# B&R Automation Studio project TD52 (part 75)

```c
  /* End of Switch: '<S7>/Switch3' */

  /* S-Function (bur_bus_in): '<Root>/Bus Input1' */
  LX2_B.BusInput1 = inst->PERM;

  /* BusSelector: '<S5>/Bus Selector7' */
  rtb_rLX2_inLimitSetup_Time = LX2_B.BusInput1.rLX2_inLimitSetup_Time;

  /* Gain: '<S7>/Gain3' incorporates:
   *  BusSelector: '<S5>/Bus Selector7'
   *  DataTypeConversion: '<S7>/Data Type Conversion2'
   *  Product: '<S7>/RateLimit_multiplier'
   */
  rtb_Gain3 = rtb_Switch7 * (real32_T)LX2_B.BusInput1.iCtrl_RateLimit_TraceBack *
    0.001F;

  /* Product: '<S41>/delta rise limit' incorporates:
   *  SampleTimeMath: '<S41>/sample time'
   *
   * About '<S41>/sample time':
   *  y = K where K = ( w * Ts )
   */
  rtb_Switch2_kt = rtb_Gain3 * 0.1F;

  /* UnitDelay: '<S7>/Unit Delay3' */
  rtb_UnitDelay3 = LX2_DWork.UnitDelay3_DSTATE;

  /* S-Function (bur_bus_in): '<Root>/Bus Input2' */
  LX2_B.BusInput2 = inst->PARA;

  /* BusSelector: '<S51>/Bus Selector4' */
  rtb_rPr_Leanox_Dev = LX2_B.BusInput.rPr_Leanox_Dev;
  rtb_rP_Set_Norm = LX2_B.BusInput.rP_Set_Norm;

  /* BusSelector: '<S51>/Bus Selector5' */
  rtb_iFiltConst_LeanoxDev_Steady =
    LX2_B.BusInput1.iFiltConst_LeanoxDev_SteadyState;
  rtb_iFiltConst_P_set_SteadyStat = LX2_B.BusInput1.iFiltConst_P_set_SteadyState;

  /* Logic: '<S51>/Logical Operator1' */
  rtb_LogicalOperator1 = !LX2_B.BusInput.bLX2_active;

  /* Outputs for Atomic SubSystem: '<S51>/Filter' */
  LX2_Filter1(rtb_iFiltConst_LeanoxDev_Steady, rtb_LogicalOperator1,
              rtb_rPr_Leanox_Dev, &LX2_B.Filter, &LX2_DWork.Filter, inst);

  /* End of Outputs for SubSystem: '<S51>/Filter' */

  /* RelationalOperator: '<S51>/ ' incorporates:
   *  Abs: '<S51>/Abs'
   *  Product: '<S51>/Thres'
   */
  rtb_u = ((real32_T)fabs(LX2_B.Filter.Switch) <=
           LX2_B.BusInput1.rThreshold_LeanoxDev_SteadyState *
           LX2_B.BusInput2.rLX2_SteadyStateFactor);

  /* Logic: '<S51>/Logical Operator3' */
  rtb_LogicalOperator3 = !LX2_B.BusInput.bLX2_active;

  /* Outputs for Atomic SubSystem: '<S51>/Filter1' */
  LX2_Filter1(rtb_iFiltConst_P_set_SteadyStat, rtb_LogicalOperator3,
              rtb_rP_Set_Norm, &LX2_B.Filter1, &LX2_DWork.Filter1, inst);

  /* End of Outputs for SubSystem: '<S51>/Filter1' */

  /* Sum: '<S51>/Sum2' */
  rtb_Switch7 = LX2_B.Filter1.Switch - rtb_rP_Set_Norm;

  /* Abs: '<S51>/Abs1' */
  rtb_Switch7 = (real32_T)fabs(rtb_Switch7);

  /* RelationalOperator: '<S51>/   ' incorporates:
   *  Product: '<S51>/Thres1'
   */
  rtb_u_b = (rtb_Switch7 <= LX2_B.BusInput1.rThreshold_P_set_SteadyState *
             LX2_B.BusInput2.rLX2_SteadyStateFactor);

  /* Logic: '<S51>/Logical Operator2' incorporates:
   *  Logic: '<S51>/Logical Operator4'
   */
  rtb_LogicalOperator2 = (LX2_B.BusInput.bLX2_active && rtb_u && rtb_u_b &&
    (!LX2_B.BusInput.bExt_SteadyState_Loss));

  /* Outputs for Atomic SubSystem: '<S51>/TON' */
  /* Logic: '<S59>/Logical Operator2' */
  rtb_LogicalOperator2_de = !rtb_LogicalOperator2;

  /* DiscreteIntegrator: '<S59>/Discrete-Time Integrator' */
  if (rtb_LogicalOperator2_de || (LX2_DWork.DiscreteTimeIntegrator_PrevRe_m != 0))
  {
    LX2_DWork.DiscreteTimeIntegrator_DSTATE_l = 0U;
  }

  /* RelationalOperator: '<S59>/Relational Operator' incorporates:
   *  DiscreteIntegrator: '<S59>/Discrete-Time Integrator'
   */
  tmp_0 = (uint32_T)LX2_DWork.DiscreteTimeIntegrator_DSTATE_l * 52429U;
  rtb_RelationalOperator_b = (((tmp_0 & 4U) != 0U) + (tmp_0 >> 3) >= ((uint32_T)
    LX2_B.BusInput1.iTiDelay_SteadyState << 16));

  /* Logic: '<S59>/Logical Operator3' */
  rtb_LogicalOperator3_e = (rtb_RelationalOperator_b && rtb_LogicalOperator2);

  /* Update for DiscreteIntegrator: '<S59>/Discrete-Time Integrator' incorporates:
   *  Logic: '<S59>/Logical Operator'
   *  Logic: '<S59>/Logical Operator1'
   */
  LX2_DWork.DiscreteTimeIntegrator_DSTATE_l = (uint16_T)((uint32_T)
    ((!rtb_RelationalOperator_b) && rtb_LogicalOperator2) + (uint32_T)
    LX2_DWork.DiscreteTimeIntegrator_DSTATE_l);
  if (rtb_LogicalOperator2_de) {
    LX2_DWork.DiscreteTimeIntegrator_PrevRe_m = 1;
  } else {
    LX2_DWork.DiscreteTimeIntegrator_PrevRe_m = 0;
  }

  /* End of Update for DiscreteIntegrator: '<S59>/Discrete-Time Integrator' */
  /* End of Outputs for SubSystem: '<S51>/TON' */

  /* MATLAB Function: '<S8>/MATLAB Function' incorporates:
   *  Constant: '<S65>/Constant'
   *  Logic: '<S52>/Logical Operator'
   *  Logic: '<S52>/Logical Operator10'
   *  RelationalOperator: '<S65>/Compare'
   */
  /* MATLAB Function 'Leanox 2.0/STM/MATLAB Function': '<S53>:1' */
  /* % Header */
  /*  This Function controls the features of LX2, like saving the map, gasmixing, enabling/disabling, timer, etc., */
  /*  depending on various inputs. */
  /*  Rev 1 : Christian Schneider, 24.08.2018 */
  /*  Rev 1.1 : Enrico Maran, 17.10.2019, Removed bLeanox_Adjust input/use */
  /*  Rev 1.2 : Enrico Maran, 17.02.2021, Removed closed loop freezing if bEng_misfire; added external interface for BPOC learning stop */
  /*  */
  /* % LX2 State Machine */
  /*  -> LEANOX 2.0 is OFF */
  if ((!LX2_B.BusInput2.bLX2_enable) || (!LX2_B.BusInput.bLX2_active)) {
    /*  LX2 off */
    /*  function undesired_operating */
    /* % function my_gasmixing <<LX2_FunReq-26>> */
    /*  define output vectors */
    /*  undefined Gastype */
    rtb_splitfactor_Gas[0] = 0.0F;
    rtb_splitfactor_Gas[1] = 0.0F;
    rtb_splitfactor_Gas[2] = 0.0F;
    rtb_splitfactor_Gas[3] = 0.0F;
    tmp[0] = 1.0F;
    tmp[1] = 1.0F;
    LX2_my_BPOC_enable_h(rtb_splitfactor_Gas, FALSE, tmp,
                         LX2_B.BusInput.bExt_BPOC_learning_Stop,
                         rtb_bBPOC_enable_a, rtb_bSave_BPOC_enable, inst);
    bCtrl_enable = FALSE;

    /*  NOx controler enable */
    bCtrl_freeze = TRUE;

    /*  freeze NOx controler output */
    b_bEng_knock = FALSE;
    bEng_misfire = FALSE;

    /*  -> LEANOX 2.0 is ON */
  } else if ((!LX2_B.BusInput.bLeanox_Engine_Man) && (rtb_LogicalOperator3_e &&
              LX2_B.BusInput.bNOx_valid && (!LX2_B.BusInput.bESC_active) &&
              (LX2_B.BusInput.rNOx_act >= 10.0F))) {
    /*  Engine in Leanox Auto Mode */
    /*              bBPOC_enable_Gas1=true;  */
    /*              bSave_BPOC_enable_Gas1=true; */
    LX2_my_gasmixing(LX2_B.BusInput.iIdx_Gtyp_Dem,
                     LX2_B.BusInput.rGT_QualMix_1_2, LX2_B.BusInput.rGT_RatioMix,
                     TRUE, LX2_B.BusInput1.rThreshold_save2map,
                     LX2_B.BusInput.bExt_BPOC_learning_Stop, rtb_splitfactor_Gas,
                     rtb_bBPOC_enable_a, rtb_bSave_BPOC_enable, inst);
    bCtrl_enable = TRUE;

    /* % function Misfire and Knocking handlig at LX2 */
    if (LX2_B.BusInput.rKnock_level <= LX2_B.BusInput1.rThreshold_knock) {
      b_bEng_knock = FALSE;
    } else {
      b_bEng_knock = TRUE;
    }

    if (LX2_B.BusInput.rMisfire_level <= LX2_B.BusInput1.rThreshold_misfire) {
      bEng_misfire = FALSE;
    } else {
      bEng_misfire = TRUE;
    }

    bCtrl_freeze = b_bEng_knock;
  } else {
    /*  Engine in Leanox Manuel Mode >or< not allowed to act -> freeze output of LX2 and do not update BPOC */
    LX2_my_gasmixing(LX2_B.BusInput.iIdx_Gtyp_Dem,
                     LX2_B.BusInput.rGT_QualMix_1_2, LX2_B.BusInput.rGT_RatioMix,
                     FALSE, LX2_B.BusInput1.rThreshold_save2map,
                     LX2_B.BusInput.bExt_BPOC_learning_Stop, rtb_splitfactor_Gas,
                     rtb_bBPOC_enable_a, rtb_bSave_BPOC_enable, inst);
    bCtrl_enable = FALSE;
    bCtrl_freeze = TRUE;
    b_bEng_knock = FALSE;
    bEng_misfire = FALSE;
  }

  /* Switch: '<S7>/Switch7' incorporates:
   *  Gain: '<S7>/mbar2bar1'
   *  MATLAB Function: '<S8>/MATLAB Function'
   */
  /* '<S53>:1:4' */
  if (bEng_misfire) {
    rtb_Switch7 = rtb_UnitDelay3;
  } else {
    rtb_Switch7 = 0.001F * LX2_B.BusInput2.rPr_LX2_OffsetLimit;
  }

  /* End of Switch: '<S7>/Switch7' */

  /* BusSelector: '<S5>/Bus Selector2' */
  rtb_Switch_nq = LX2_B.BusInput2.rLX2_Ctrl_Tn;

  /* RelationalOperator: '<S32>/Compare' incorporates:
   *  BusSelector: '<S5>/Bus Selector2'
   *  Constant: '<S32>/Constant'
   */
  rtb_Compare_n = (LX2_B.BusInput2.rLX2_Ctrl_Tn <= 0.0F);

  /* BusSelector: '<S5>/Bus Selector4' */
  rtb_rNOx_act_g = LX2_B.BusInput.rNOx_act;

  /* Logic: '<S5>/Logical Operator6' */
  rtb_LogicalOperator6_a = !LX2_B.BusInput.bLX2_active;

  /* UnitDelay: '<S7>/Unit Delay1' */
  rtb_UnitDelay1 = LX2_DWork.UnitDelay1_DSTATE;

  /* Logic: '<S52>/Logical Operator11' incorporates:
   *  Logic: '<S52>/Logical Operator5'
   *  Logic: '<S52>/Logical Operator6'
   *  Logic: '<S52>/Logical Operator7'
   *  Logic: '<S52>/Logical Operator8'
   *  UnitDelay: '<S52>/Unit Delay1'
   */
  rtb_LogicalOperator_f = (LX2_DWork.UnitDelay1_DSTATE_l ||
    (((!LX2_B.BusInput2.bLX2_enable) || (!LX2_B.BusInput.bLX2_active)) &&
     LX2_B.BusInput.bBPOC_reset));

  /* Logic: '<S54>/Logical Operator4' incorporates:
   *  Logic: '<S54>/Logical Operator1'
   *  Logic: '<S54>/Logical Operator27'
   *  Logic: '<S54>/Logical Operator3'
   *  UnitDelay: '<S54>/Unit Delay'
   */
  rtb_LogicalOperator4_n = ((!LX2_DWork.UnitDelay_DSTATE_l) &&
    (!rtb_LogicalOperator_f) && (rtb_bSave_BPOC_enable[0] ||
    rtb_bSave_BPOC_enable[1] || rtb_bSave_BPOC_enable[2] ||
    rtb_bSave_BPOC_enable[3]));

  /* DataTypeConversion: '<S54>/Data Type Conversion' incorporates:
   *  BusSelector: '<S54>/Bus Selector5'
   */
  rtb_DataTypeConversion = (real32_T)LX2_B.BusInput1.iTiUpdate_BPOC;

  /* Outputs for Atomic SubSystem: '<S54>/TON' */
  LX2_TON(rtb_LogicalOperator4_n, rtb_DataTypeConversion, &LX2_B.TON_p,
          &LX2_DWork.TON_p, inst);

  /* End of Outputs for SubSystem: '<S54>/TON' */

  /* Switch: '<S54>/Switch2' incorporates:
   *  Switch: '<S54>/Switch1'
   */
  if (rtb_LogicalOperator_f) {
    rtb_Switch2_a_idx = TRUE;
    rtb_Switch2_a_idx_0 = TRUE;
    rtb_Switch2_a_idx_1 = TRUE;
    rtb_Switch2_a_idx_2 = TRUE;
  } else if (LX2_B.TON_p.LogicalOperator3) {
    /* Switch: '<S54>/Switch1' */
    rtb_Switch2_a_idx = rtb_bSave_BPOC_enable[0];
    rtb_Switch2_a_idx_0 = rtb_bSave_BPOC_enable[1];
    rtb_Switch2_a_idx_1 = rtb_bSave_BPOC_enable[2];
    rtb_Switch2_a_idx_2 = rtb_bSave_BPOC_enable[3];
  } else {
    rtb_Switch2_a_idx = FALSE;
    rtb_Switch2_a_idx_0 = FALSE;
    rtb_Switch2_a_idx_1 = FALSE;
    rtb_Switch2_a_idx_2 = FALSE;
  }

  /* End of Switch: '<S54>/Switch2' */

  /* Gain: '<S8>/Gain7' */
  rtb_Gain7 = 100.0F * LX2_B.BusInput.rP_Set_Norm;

  /* BusSelector: '<S8>/Bus Selector4' */
  rtb_iFilterConst_P_set = LX2_B.BusInput1.iFilterConst_P_set;

  /* Logic: '<S8>/Logical Operator8' */
  rtb_LogicalOperator8_g = !LX2_B.BusInput.bLX2_active;

  /* Outputs for Atomic SubSystem: '<S8>/Filter1' */
  LX2_Filter1(rtb_iFilterConst_P_set, rtb_LogicalOperator8_g, rtb_Gain7,
              &LX2_B.Filter1_i, &LX2_DWork.Filter1_i, inst);

  /* End of Outputs for SubSystem: '<S8>/Filter1' */

  /* Gain: '<S10>/mbar2bar' */
  rtb_UnitDelay3 = 0.001F * LX2_B.BusInput2.rPr_LX2_OffsetLimit;

  /* Logic: '<S10>/Logical Operator7' incorporates:
   *  Logic: '<S10>/Logical Operator8'
   *  Selector: '<S10>/Selector1'
   */
  rtb_LogicalOperator7_m = ((!rtb_LogicalOperator_f) && rtb_bSave_BPOC_enable[0]);

  /* Logic: '<S10>/Logical Operator2' incorporates:
   *  Logic: '<S10>/Logical Operator3'
   */
  rtb_RelationalOperator_b = ((!rtb_LogicalOperator7_m) || rtb_LogicalOperator_f);

  /* BusSelector: '<S6>/Bus Selector6' */
  for (i = 0; i < 5; i++) {
    rtb_rP_Lp_c[i] = LX2_B.BusInput.rP_Nom[i];
    rtb_rPr_LX2_offset_Lp_c[i] = LX2_B.BusInput.rP_Lp_b[i];
    rtb_rPr_LX2_offset_Lp_a[i] = LX2_B.BusInput.rP_Lp_a[i];
    rtb_rPr_LX2_offset_Lp_b[i] = LX2_B.BusInput.rP_Lp_c[i];
  }

  rtb_bLp_c_ena = LX2_B.BusInput.bLp_c_ena;

  /* End of BusSelector: '<S6>/Bus Selector6' */

  /* Logic: '<S10>/Logical Operator5' */
  rtb_LogicalOperator5_k = !rtb_LogicalOperator_f;

  /* Delay: '<S10>/Delay2' */
  didZcEventOccur = (((LX2_PrevZCSigState.Delay2_Reset_ZCE == LX2_POS_ZCSIG) !=
                      rtb_RelationalOperator_b) &&
                     (LX2_PrevZCSigState.Delay2_Reset_ZCE !=
                      LX2_UNINITIALIZED_ZCSIG));
  LX2_PrevZCSigState.Delay2_Reset_ZCE = (uint8_T)rtb_RelationalOperator_b;
  if (rtb_RelationalOperator_b || didZcEventOccur) {
    LX2_DWork.icLoad = 1U;
  }

  for (i = 0; i < 11; i++) {
    if (LX2_DWork.icLoad != 0) {
      /* Switch: '<S10>/Switch5' incorporates:
       *  Constant: '<S10>/Constant5'
       */
      if (rtb_LogicalOperator5_k) {
        LX2_DWork.Delay2_DSTATE[i] = LX2_B.BusInput.rLX2_BPOC_Gas1[i];
      } else {
        LX2_DWork.Delay2_DSTATE[i] = 0.0F;
      }

      /* End of Switch: '<S10>/Switch5' */
    }

    rtb_Delay2[i] = LX2_DWork.Delay2_DSTATE[i];
  }

  /* End of Delay: '<S10>/Delay2' */
  /* Dynamic Look-Up Table Block: '<S10>/Interpolate BPOC_actual'
   * Input0  Data Type:  Floating Point real32_T
   * Input1  Data Type:  Floating Point real32_T
   * Input2  Data Type:  Floating Point real32_T
   * Output0 Data Type:  Floating Point real32_T
   * Lookup Method: Linear_Endpoint
   *
   */
  LookUp_real32_T_real32_T( &(rtb_Selector12), rtb_Delay2,
    LX2_B.Filter1_i.Switch, LX2_ConstP.pooled14, 10U, inst);

  /* UnitDelay: '<S6>/Unit Delay2' */
  rtb_UnitDelay2 = LX2_DWork.UnitDelay2_DSTATE;

  /* Sum: '<S10>/Sum1' incorporates:
   *  Product: '<S10>/Divide4'
   *  Selector: '<S10>/Selector2'
   *  Sum: '<S10>/Sum2'
   *  UnitDelay: '<S6>/Unit Delay2'
   */
  rtb_Sum1 = (LX2_DWork.UnitDelay2_DSTATE - rtb_Selector12) *
    rtb_splitfactor_Gas[0] + rtb_Selector12;

  /* Logic: '<S10>/Logical Operator6' incorporates:
   *  Logic: '<S10>/Logical Operator4'
   */
  rtb_RelationalOperator_b = ((!rtb_LogicalOperator7_m) || rtb_LogicalOperator_f);

  /* Logic: '<S10>/Logical Operator1' */
  rtb_LogicalOperator5_k = !rtb_LogicalOperator_f;

  /* Delay: '<S10>/Delay1' */
  didZcEventOccur = (((LX2_PrevZCSigState.Delay1_Reset_ZCE == LX2_POS_ZCSIG) !=
                      rtb_RelationalOperator_b) &&
                     (LX2_PrevZCSigState.Delay1_Reset_ZCE !=
                      LX2_UNINITIALIZED_ZCSIG));
  LX2_PrevZCSigState.Delay1_Reset_ZCE = (uint8_T)rtb_RelationalOperator_b;
  if (rtb_RelationalOperator_b || didZcEventOccur) {
    LX2_DWork.icLoad_o = 1U;
  }

  for (i = 0; i < 11; i++) {
    if (LX2_DWork.icLoad_o != 0) {
      /* Switch: '<S10>/Switch4' incorporates:
       *  Constant: '<S10>/Constant4'
       */
      if (rtb_LogicalOperator5_k) {
        LX2_DWork.Delay1_DSTATE[i] = LX2_B.BusInput.bLX2_BPOC_measured_Gas1[i];
      } else {
        LX2_DWork.Delay1_DSTATE[i] = FALSE;
      }

      /* End of Switch: '<S10>/Switch4' */
    }

    rtb_Delay1[i] = LX2_DWork.Delay1_DSTATE[i];
  }

  /* End of Delay: '<S10>/Delay1' */

  /* Selector: '<S10>/Selector6' incorporates:
   *  Constant: '<S6>/Constant3'
   */
  rtb_Selector12 = rtb_rPr_LX2_offset_Lp_c[1];

  /* Selector: '<S10>/Selector4' incorporates:
   *  Constant: '<S6>/Constant3'
   */
  rtb_Switch2_b = rtb_rP_Lp_c[1];

  /* Abs: '<S16>/Abs' */
  rtb_Abs = (real32_T)fabs(rtb_Switch2_b);

  /* Switch: '<S16>/Switch' incorporates:
   *  RelationalOperator: '<S16>/Relational Operator'
   */
  if (2.22044605E-16F >= rtb_Abs) {
    rtb_Switch2_b = 2.22044605E-16F;
  }

  /* End of Switch: '<S16>/Switch' */

  /* Gain: '<S10>/Gain1' incorporates:
   *  Constant: '<S6>/Constant3'
   *  Product: '<S10>/Divide'
   *  Selector: '<S10>/Selector12'
   *  Selector: '<S10>/Selector5'
   */
  rtb_Lp2Lp3Lp_c[0] = rtb_Selector12 / rtb_Switch2_b * 100.0F;
  rtb_Lp2Lp3Lp_c[1] = rtb_rPr_LX2_offset_Lp_a[1] / rtb_Switch2_b * 100.0F;
  rtb_Lp2Lp3Lp_c[2] = rtb_rPr_LX2_offset_Lp_b[1] / rtb_Switch2_b * 100.0F;

  /* Gain: '<S6>/SlopeMax_factor' */
  rtb_Abs = 0.01F * LX2_B.BusInput2.rPr_LX2_OffsetLimit;

  /* Gain: '<S10>/mbar2bar2' */
  rtb_mbar2bar2 = 0.001F * rtb_Abs;

  /* Gain: '<S6>/SlopeMaxEx_factor' */
  rtb_Switch2_b = 0.003F * LX2_B.BusInput2.rPr_LX2_OffsetLimit;

  /* Gain: '<S10>/mbar2bar3' */
  rtb_mbar2bar3 = 0.001F * rtb_Switch2_b;

  /* BusSelector: '<S6>/Bus Selector5' */
  rtb_iWeight_Lp_0kW = LX2_B.BusInput1.iWeight_Lp_0kW;
  rtb_iWeight_Lp_b = LX2_B.BusInput1.iWeight_Lp_b;
  rtb_iWeight_Lp_a = LX2_B.BusInput1.iWeight_Lp_a;
  rtb_iWeight_Lp_c = LX2_B.BusInput1.iWeight_Lp_c;

  /* Gain: '<S10>/mbar2bar4' */
  rtb_mbar2bar4 = 0.001F * LX2_B.BusInput2.rPr_LX2_OffsetLimit;

  /* MATLAB Function: '<S10>/Boost Pressure Offset Curve' */
  LX2_BoostPressureOffsetCurve(LX2_B.Filter1_i.Switch, rtb_Sum1, rtb_Delay2,
    rtb_Delay1, rtb_Lp2Lp3Lp_c, rtb_bLp_c_ena, rtb_mbar2bar2, rtb_mbar2bar3,
    rtb_iWeight_Lp_0kW, rtb_iWeight_Lp_b, rtb_iWeight_Lp_a, rtb_iWeight_Lp_c,
    rtb_mbar2bar4, rtb_LogicalOperator7_m, &LX2_B.sf_BoostPressureOffsetCurve, inst);

  /* Gain: '<S5>/LowerLimit_factor' */
  rtb_LowerLimit_factor = -LX2_B.BusInput2.rPr_LX2_OffsetLimit;

  /* Gain: '<S10>/mbar2bar1' incorporates:
   *  Gain: '<S5>/LowerLimit_factor'
   */
  rtb_Switch3 = 0.001F * -LX2_B.BusInput2.rPr_LX2_OffsetLimit;
  for (i = 0; i < 11; i++) {
    /* Switch: '<S17>/Switch2' incorporates:
     *  RelationalOperator: '<S17>/LowerRelop1'
     *  RelationalOperator: '<S17>/UpperRelop'
     *  Switch: '<S17>/Switch'
     */
    if (LX2_B.sf_BoostPressureOffsetCurve.OUT_offset[i] > rtb_UnitDelay3) {
      rtb_splitfactor_VISU_idx = rtb_UnitDelay3;
    } else if (LX2_B.sf_BoostPressureOffsetCurve.OUT_offset[i] < rtb_Switch3) {
      /* Switch: '<S17>/Switch' */
      rtb_splitfactor_VISU_idx = rtb_Switch3;
    } else {
      rtb_splitfactor_VISU_idx = LX2_B.sf_BoostPressureOffsetCurve.OUT_offset[i];
    }

    /* Switch: '<S10>/Switch1' incorporates:
     *  Selector: '<S10>/Selector7'
     */
    if (rtb_Switch2_a_idx) {
      rtb_Switch1[i] = rtb_splitfactor_VISU_idx;
    } else {
      rtb_Switch1[i] = LX2_B.BusInput.rLX2_BPOC_Gas1[i];
    }

    /* End of Switch: '<S10>/Switch1' */

    /* Switch: '<S17>/Switch2' */
    rtb_Switch2[i] = rtb_splitfactor_VISU_idx;
  }

  /* Switch: '<S10>/Switch3' incorporates:
   *  Constant: '<S10>/Constant2'
   *  Constant: '<S10>/Constant3'
   *  Selector: '<S10>/Selector3'
   */
  if (rtb_bBPOC_enable_a[0]) {
    /* Dynamic Look-Up Table Block: '<S10>/Interpolate BPOC'
     * Input0  Data Type:  Floating Point real32_T
     * Input1  Data Type:  Floating Point real32_T
     * Input2  Data Type:  Floating Point real32_T
     * Output0 Data Type:  Floating Point real32_T
     * Lookup Method: Linear_Endpoint
     *
     */
    LookUp_real32_T_real32_T( &(rtb_InterpolateBPOC_a), rtb_Switch1,
      LX2_B.Filter1_i.Switch, LX2_ConstP.pooled14, 10U, inst);
    rtb_Switch3 = rtb_InterpolateBPOC_a;
  } else {
    rtb_Switch3 = 0.0F;
  }

  /* End of Switch: '<S10>/Switch3' */

  /* Gain: '<S11>/mbar2bar' */
  rtb_UnitDelay3 = 0.001F * LX2_B.BusInput2.rPr_LX2_OffsetLimit;

  /* Logic: '<S11>/Logical Operator7' incorporates:
   *  Logic: '<S11>/Logical Operator8'
   *  Selector: '<S11>/Selector1'
   */
  rtb_LogicalOperator7_e = ((!rtb_LogicalOperator_f) && rtb_bSave_BPOC_enable[1]);

  /* Logic: '<S11>/Logical Operator2' incorporates:
   *  Logic: '<S11>/Logical Operator3'
   */
  rtb_RelationalOperator_b = ((!rtb_LogicalOperator7_e) || rtb_LogicalOperator_f);

  /* BusSelector: '<S6>/Bus Selector8' */
  for (i = 0; i < 5; i++) {
    rtb_rPr_LX2_offset_Lp_b[i] = LX2_B.BusInput.rP_Nom[i];
    rtb_rPr_LX2_offset_Lp_a[i] = LX2_B.BusInput.rP_Lp_b[i];
    rtb_rPr_LX2_offset_Lp_c[i] = LX2_B.BusInput.rP_Lp_a[i];
    rtb_rP_Lp_c[i] = LX2_B.BusInput.rP_Lp_c[i];
  }

  rtb_bLp_c_ena_i = LX2_B.BusInput.bLp_c_ena;

  /* End of BusSelector: '<S6>/Bus Selector8' */

  /* Logic: '<S11>/Logical Operator5' */
  rtb_LogicalOperator5_k = !rtb_LogicalOperator_f;

  /* Delay: '<S11>/Delay2' */
  didZcEventOccur = (((LX2_PrevZCSigState.Delay2_Reset_ZCE_o == LX2_POS_ZCSIG)
                      != rtb_RelationalOperator_b) &&
                     (LX2_PrevZCSigState.Delay2_Reset_ZCE_o !=
                      LX2_UNINITIALIZED_ZCSIG));
  LX2_PrevZCSigState.Delay2_Reset_ZCE_o = (uint8_T)rtb_RelationalOperator_b;
  if (rtb_RelationalOperator_b || didZcEventOccur) {
    LX2_DWork.icLoad_or = 1U;
  }

  for (i = 0; i < 11; i++) {
    if (LX2_DWork.icLoad_or != 0) {
      /* Switch: '<S11>/Switch5' incorporates:
       *  Constant: '<S11>/Constant5'
       */
      if (rtb_LogicalOperator5_k) {
        LX2_DWork.Delay2_DSTATE_j[i] = LX2_B.BusInput.rLX2_BPOC_Gas2[i];
      } else {
        LX2_DWork.Delay2_DSTATE_j[i] = 0.0F;
      }

      /* End of Switch: '<S11>/Switch5' */
    }

    rtb_Delay2_e[i] = LX2_DWork.Delay2_DSTATE_j[i];
  }

  /* End of Delay: '<S11>/Delay2' */
  /* Dynamic Look-Up Table Block: '<S11>/Interpolate BPOC_actual'
   * Input0  Data Type:  Floating Point real32_T
   * Input1  Data Type:  Floating Point real32_T
   * Input2  Data Type:  Floating Point real32_T
   * Output0 Data Type:  Floating Point real32_T
   * Lookup Method: Linear_Endpoint
   *
   */
  LookUp_real32_T_real32_T( &(rtb_Selector12), rtb_Delay2_e,
    LX2_B.Filter1_i.Switch, LX2_ConstP.pooled14, 10U, inst);

  /* Sum: '<S11>/Sum1' incorporates:
   *  Product: '<S11>/Divide4'
   *  Selector: '<S11>/Selector2'
   *  Sum: '<S11>/Sum2'
   */
  rtb_Sum1_e = (rtb_UnitDelay2 - rtb_Selector12) * rtb_splitfactor_Gas[1] +
    rtb_Selector12;

  /* Logic: '<S11>/Logical Operator6' incorporates:
   *  Logic: '<S11>/Logical Operator4'
   */
  rtb_RelationalOperator_b = ((!rtb_LogicalOperator7_e) || rtb_LogicalOperator_f);

  /* Logic: '<S11>/Logical Operator1' */
  rtb_LogicalOperator5_k = !rtb_LogicalOperator_f;

  /* Delay: '<S11>/Delay1' */
  didZcEventOccur = (((LX2_PrevZCSigState.Delay1_Reset_ZCE_n == LX2_POS_ZCSIG)
                      != rtb_RelationalOperator_b) &&
                     (LX2_PrevZCSigState.Delay1_Reset_ZCE_n !=
                      LX2_UNINITIALIZED_ZCSIG));
  LX2_PrevZCSigState.Delay1_Reset_ZCE_n = (uint8_T)rtb_RelationalOperator_b;
  if (rtb_RelationalOperator_b || didZcEventOccur) {
    LX2_DWork.icLoad_oj = 1U;
  }

  for (i = 0; i < 11; i++) {
    if (LX2_DWork.icLoad_oj != 0) {
      /* Switch: '<S11>/Switch4' incorporates:
       *  Constant: '<S11>/Constant4'
       */
      if (rtb_LogicalOperator5_k) {
        LX2_DWork.Delay1_DSTATE_l[i] = LX2_B.BusInput.bLX2_BPOC_measured_Gas2[i];
      } else {
        LX2_DWork.Delay1_DSTATE_l[i] = FALSE;
      }

      /* End of Switch: '<S11>/Switch4' */
    }

    rtb_Delay1_g[i] = LX2_DWork.Delay1_DSTATE_l[i];
  }

  /* End of Delay: '<S11>/Delay1' */

  /* Selector: '<S11>/Selector6' incorporates:
   *  Constant: '<S6>/Constant1'
   */
  rtb_Selector12 = rtb_rPr_LX2_offset_Lp_a[2];

  /* Selector: '<S11>/Selector12' incorporates:
   *  Constant: '<S6>/Constant1'
   */
  rtb_Divide = rtb_rP_Lp_c[2];

  /* Selector: '<S11>/Selector4' incorporates:
   *  Constant: '<S6>/Constant1'
   */
  rtb_Switch2_l = rtb_rPr_LX2_offset_Lp_b[2];

  /* Switch: '<S20>/Switch' incorporates:
   *  Abs: '<S20>/Abs'
   *  RelationalOperator: '<S20>/Relational Operator'
   */
  if (2.22044605E-16F >= (real32_T)fabs(rtb_Switch2_l)) {
    rtb_Switch2_l = 2.22044605E-16F;
  }

  /* End of Switch: '<S20>/Switch' */

  /* Gain: '<S11>/Gain1' incorporates:
   *  Constant: '<S6>/Constant1'
   *  Product: '<S11>/Divide'
   *  Selector: '<S11>/Selector5'
   */
  rtb_Lp2Lp3Lp_c_n[0] = rtb_Selector12 / rtb_Switch2_l * 100.0F;
  rtb_Lp2Lp3Lp_c_n[1] = rtb_rPr_LX2_offset_Lp_c[2] / rtb_Switch2_l * 100.0F;
  rtb_Lp2Lp3Lp_c_n[2] = rtb_Divide / rtb_Switch2_l * 100.0F;

  /* Gain: '<S11>/mbar2bar2' */
  rtb_mbar2bar2_e = 0.001F * rtb_Abs;

  /* Gain: '<S11>/mbar2bar3' */
  rtb_mbar2bar3_h = 0.001F * rtb_Switch2_b;

  /* BusSelector: '<S6>/Bus Selector7' */
  rtb_iWeight_Lp_0kW_e = LX2_B.BusInput1.iWeight_Lp_0kW;
  rtb_iWeight_Lp_b_c = LX2_B.BusInput1.iWeight_Lp_b;
  rtb_iWeight_Lp_a_m = LX2_B.BusInput1.iWeight_Lp_a;
  rtb_iWeight_Lp_c_m = LX2_B.BusInput1.iWeight_Lp_c;

  /* Gain: '<S11>/mbar2bar4' */
  rtb_mbar2bar4_m = 0.001F * LX2_B.BusInput2.rPr_LX2_OffsetLimit;

  /* MATLAB Function: '<S11>/Boost Pressure Offset Curve' */
  LX2_BoostPressureOffsetCurve(LX2_B.Filter1_i.Switch, rtb_Sum1_e, rtb_Delay2_e,
    rtb_Delay1_g, rtb_Lp2Lp3Lp_c_n, rtb_bLp_c_ena_i, rtb_mbar2bar2_e,
    rtb_mbar2bar3_h, rtb_iWeight_Lp_0kW_e, rtb_iWeight_Lp_b_c,
    rtb_iWeight_Lp_a_m, rtb_iWeight_Lp_c_m, rtb_mbar2bar4_m,
    rtb_LogicalOperator7_e, &LX2_B.sf_BoostPressureOffsetCurve_f, inst);

  /* Gain: '<S11>/mbar2bar1' */
  rtb_SumofElements2 = 0.001F * rtb_LowerLimit_factor;
  for (i = 0; i < 11; i++) {
    /* Switch: '<S21>/Switch2' incorporates:
     *  RelationalOperator: '<S21>/LowerRelop1'
     *  RelationalOperator: '<S21>/UpperRelop'
     *  Switch: '<S21>/Switch'
     */
    if (LX2_B.sf_BoostPressureOffsetCurve_f.OUT_offset[i] > rtb_UnitDelay3) {
      rtb_splitfactor_VISU_idx = rtb_UnitDelay3;
    } else if (LX2_B.sf_BoostPressureOffsetCurve_f.OUT_offset[i] <
               rtb_SumofElements2) {
      /* Switch: '<S21>/Switch' */
      rtb_splitfactor_VISU_idx = rtb_SumofElements2;
    } else {
      rtb_splitfactor_VISU_idx =
        LX2_B.sf_BoostPressureOffsetCurve_f.OUT_offset[i];
    }

    /* Switch: '<S11>/Switch1' incorporates:
     *  Selector: '<S11>/Selector7'
     */
    if (rtb_Switch2_a_idx_0) {
      rtb_Switch1_m[i] = rtb_splitfactor_VISU_idx;
    } else {
      rtb_Switch1_m[i] = LX2_B.BusInput.rLX2_BPOC_Gas2[i];
    }

    /* End of Switch: '<S11>/Switch1' */

    /* Switch: '<S21>/Switch2' */
    rtb_Switch2_j[i] = rtb_splitfactor_VISU_idx;
  }

  /* Switch: '<S11>/Switch3' incorporates:
   *  Constant: '<S11>/Constant2'
   *  Constant: '<S11>/Constant3'
   *  Selector: '<S11>/Selector3'
   */
  if (rtb_bBPOC_enable_a[1]) {
    /* Dynamic Look-Up Table Block: '<S11>/Interpolate BPOC'
     * Input0  Data Type:  Floating Point real32_T
     * Input1  Data Type:  Floating Point real32_T
     * Input2  Data Type:  Floating Point real32_T
     * Output0 Data Type:  Floating Point real32_T
     * Lookup Method: Linear_Endpoint
     *
     */
    LookUp_real32_T_real32_T( &(rtb_InterpolateBPOC_h), rtb_Switch1_m,
      LX2_B.Filter1_i.Switch, LX2_ConstP.pooled14, 10U, inst);
    rtb_SumofElements2 = rtb_InterpolateBPOC_h;
  } else {
    rtb_SumofElements2 = 0.0F;
  }

  /* End of Switch: '<S11>/Switch3' */

  /* Gain: '<S12>/mbar2bar' */
  rtb_Switch2_l = 0.001F * LX2_B.BusInput2.rPr_LX2_OffsetLimit;

  /* Logic: '<S12>/Logical Operator7' incorporates:
   *  Logic: '<S12>/Logical Operator8'
   *  Selector: '<S12>/Selector1'
   */
  rtb_LogicalOperator7_l = ((!rtb_LogicalOperator_f) && rtb_bSave_BPOC_enable[2]);

  /* Logic: '<S12>/Logical Operator2' incorporates:
   *  Logic: '<S12>/Logical Operator3'
   */
  rtb_RelationalOperator_b = ((!rtb_LogicalOperator7_l) || rtb_LogicalOperator_f);

  /* BusSelector: '<S6>/Bus Selector10' */
  for (i = 0; i < 5; i++) {
    rtb_rPr_LX2_offset_Lp_b[i] = LX2_B.BusInput.rP_Nom[i];
    rtb_rPr_LX2_offset_Lp_a[i] = LX2_B.BusInput.rP_Lp_b[i];
    rtb_rPr_LX2_offset_Lp_c[i] = LX2_B.BusInput.rP_Lp_a[i];
    rtb_rP_Lp_c[i] = LX2_B.BusInput.rP_Lp_c[i];
  }

  rtb_bLp_c_ena_h = LX2_B.BusInput.bLp_c_ena;

  /* End of BusSelector: '<S6>/Bus Selector10' */

  /* Logic: '<S12>/Logical Operator5' */
  rtb_LogicalOperator5_k = !rtb_LogicalOperator_f;

  /* Delay: '<S12>/Delay2' */
  didZcEventOccur = (((LX2_PrevZCSigState.Delay2_Reset_ZCE_or == LX2_POS_ZCSIG)
                      != rtb_RelationalOperator_b) &&
                     (LX2_PrevZCSigState.Delay2_Reset_ZCE_or !=
                      LX2_UNINITIALIZED_ZCSIG));
  LX2_PrevZCSigState.Delay2_Reset_ZCE_or = (uint8_T)rtb_RelationalOperator_b;
  if (rtb_RelationalOperator_b || didZcEventOccur) {
    LX2_DWork.icLoad_p = 1U;
  }

  for (i = 0; i < 11; i++) {
    if (LX2_DWork.icLoad_p != 0) {
      /* Switch: '<S12>/Switch5' incorporates:
       *  Constant: '<S12>/Constant5'
       */
      if (rtb_LogicalOperator5_k) {
        LX2_DWork.Delay2_DSTATE_b[i] = LX2_B.BusInput.rLX2_BPOC_Gas3[i];
      } else {
        LX2_DWork.Delay2_DSTATE_b[i] = 0.0F;
      }

      /* End of Switch: '<S12>/Switch5' */
    }

    rtb_Delay2_o[i] = LX2_DWork.Delay2_DSTATE_b[i];
  }

  /* End of Delay: '<S12>/Delay2' */
  /* Dynamic Look-Up Table Block: '<S12>/Interpolate BPOC_actual'
   * Input0  Data Type:  Floating Point real32_T
   * Input1  Data Type:  Floating Point real32_T
   * Input2  Data Type:  Floating Point real32_T
   * Output0 Data Type:  Floating Point real32_T
   * Lookup Method: Linear_Endpoint
   *
   */
  LookUp_real32_T_real32_T( &(rtb_Divide), rtb_Delay2_o, LX2_B.Filter1_i.Switch,
    LX2_ConstP.pooled14, 10U, inst);

  /* Sum: '<S12>/Sum1' incorporates:
   *  Product: '<S12>/Divide4'
   *  Selector: '<S12>/Selector2'
   *  Sum: '<S12>/Sum2'
   */
  rtb_Sum1_b = (rtb_UnitDelay2 - rtb_Divide) * rtb_splitfactor_Gas[2] +
    rtb_Divide;

  /* Logic: '<S12>/Logical Operator6' incorporates:
   *  Logic: '<S12>/Logical Operator4'
   */
  rtb_RelationalOperator_b = ((!rtb_LogicalOperator7_l) || rtb_LogicalOperator_f);

  /* Logic: '<S12>/Logical Operator1' */
  rtb_LogicalOperator5_k = !rtb_LogicalOperator_f;

  /* Delay: '<S12>/Delay1' */
  didZcEventOccur = (((LX2_PrevZCSigState.Delay1_Reset_ZCE_e == LX2_POS_ZCSIG)
                      != rtb_RelationalOperator_b) &&
                     (LX2_PrevZCSigState.Delay1_Reset_ZCE_e !=
                      LX2_UNINITIALIZED_ZCSIG));
  LX2_PrevZCSigState.Delay1_Reset_ZCE_e = (uint8_T)rtb_RelationalOperator_b;
  if (rtb_RelationalOperator_b || didZcEventOccur) {
    LX2_DWork.icLoad_d = 1U;
  }

  for (i = 0; i < 11; i++) {
    if (LX2_DWork.icLoad_d != 0) {
      /* Switch: '<S12>/Switch4' incorporates:
       *  Constant: '<S12>/Constant4'
       */
      if (rtb_LogicalOperator5_k) {
        LX2_DWork.Delay1_DSTATE_o[i] = LX2_B.BusInput.bLX2_BPOC_measured_Gas3[i];
      } else {
        LX2_DWork.Delay1_DSTATE_o[i] = FALSE;
      }

      /* End of Switch: '<S12>/Switch4' */
    }

    rtb_Delay1_l[i] = LX2_DWork.Delay1_DSTATE_o[i];
  }

  /* End of Delay: '<S12>/Delay1' */

  /* Selector: '<S12>/Selector6' incorporates:
   *  Constant: '<S6>/Constant5'
   */
  rtb_Divide = rtb_rPr_LX2_offset_Lp_a[3];

  /* Selector: '<S12>/Selector12' incorporates:
   *  Constant: '<S6>/Constant5'
   */
  rtb_Selector12 = rtb_rP_Lp_c[3];

  /* Switch: '<S24>/Switch' incorporates:
   *  Abs: '<S24>/Abs'
   *  Constant: '<S6>/Constant5'
   *  RelationalOperator: '<S24>/Relational Operator'
   *  Selector: '<S12>/Selector4'
   */
  if (2.22044605E-16F >= (real32_T)fabs(rtb_rPr_LX2_offset_Lp_b[3])) {
    rtb_UnitDelay3 = 2.22044605E-16F;
  } else {
    rtb_UnitDelay3 = rtb_rPr_LX2_offset_Lp_b[3];
  }

  /* End of Switch: '<S24>/Switch' */

  /* Gain: '<S12>/Gain1' incorporates:
   *  Constant: '<S6>/Constant5'
   *  Product: '<S12>/Divide'
   *  Selector: '<S12>/Selector5'
   */
  rtb_Lp2Lp3Lp_c_l[0] = rtb_Divide / rtb_UnitDelay3 * 100.0F;
  rtb_Lp2Lp3Lp_c_l[1] = rtb_rPr_LX2_offset_Lp_c[3] / rtb_UnitDelay3 * 100.0F;
  rtb_Lp2Lp3Lp_c_l[2] = rtb_Selector12 / rtb_UnitDelay3 * 100.0F;

  /* Gain: '<S12>/mbar2bar2' */
  rtb_mbar2bar2_o = 0.001F * rtb_Abs;

  /* Gain: '<S12>/mbar2bar3' */
  rtb_mbar2bar3_o = 0.001F * rtb_Switch2_b;

  /* BusSelector: '<S6>/Bus Selector9' */
  rtb_iWeight_Lp_0kW_d = LX2_B.BusInput1.iWeight_Lp_0kW;
  rtb_iWeight_Lp_b_a = LX2_B.BusInput1.iWeight_Lp_b;
  rtb_iWeight_Lp_a_j = LX2_B.BusInput1.iWeight_Lp_a;
  rtb_iWeight_Lp_c_f = LX2_B.BusInput1.iWeight_Lp_c;

  /* Gain: '<S12>/mbar2bar4' */
  rtb_mbar2bar4_e = 0.001F * LX2_B.BusInput2.rPr_LX2_OffsetLimit;

  /* MATLAB Function: '<S12>/Boost Pressure Offset Curve' */
  LX2_BoostPressureOffsetCurve(LX2_B.Filter1_i.Switch, rtb_Sum1_b, rtb_Delay2_o,
    rtb_Delay1_l, rtb_Lp2Lp3Lp_c_l, rtb_bLp_c_ena_h, rtb_mbar2bar2_o,
    rtb_mbar2bar3_o, rtb_iWeight_Lp_0kW_d, rtb_iWeight_Lp_b_a,
    rtb_iWeight_Lp_a_j, rtb_iWeight_Lp_c_f, rtb_mbar2bar4_e,
    rtb_LogicalOperator7_l, &LX2_B.sf_BoostPressureOffsetCurve_d, inst);

  /* Gain: '<S12>/mbar2bar1' */
  rtb_SumofElements1 = 0.001F * rtb_LowerLimit_factor;
  for (i = 0; i < 11; i++) {
    /* Switch: '<S25>/Switch2' incorporates:
     *  RelationalOperator: '<S25>/LowerRelop1'
     *  RelationalOperator: '<S25>/UpperRelop'
     *  Switch: '<S25>/Switch'
     */
    if (LX2_B.sf_BoostPressureOffsetCurve_d.OUT_offset[i] > rtb_Switch2_l) {
      rtb_splitfactor_VISU_idx = rtb_Switch2_l;
    } else if (LX2_B.sf_BoostPressureOffsetCurve_d.OUT_offset[i] <
               rtb_SumofElements1) {
      /* Switch: '<S25>/Switch' */
      rtb_splitfactor_VISU_idx = rtb_SumofElements1;
    } else {
      rtb_splitfactor_VISU_idx =
        LX2_B.sf_BoostPressureOffsetCurve_d.OUT_offset[i];
    }

    /* Switch: '<S12>/Switch1' incorporates:
     *  Selector: '<S12>/Selector7'
     */
    if (rtb_Switch2_a_idx_1) {
      rtb_Switch1_i[i] = rtb_splitfactor_VISU_idx;
    } else {
      rtb_Switch1_i[i] = LX2_B.BusInput.rLX2_BPOC_Gas3[i];
    }

    /* End of Switch: '<S12>/Switch1' */

    /* Switch: '<S25>/Switch2' */
    rtb_Switch2_k[i] = rtb_splitfactor_VISU_idx;
  }

  /* Switch: '<S12>/Switch3' incorporates:
   *  Constant: '<S12>/Constant2'
   *  Constant: '<S12>/Constant3'
   *  Selector: '<S12>/Selector3'
   */
  if (rtb_bBPOC_enable_a[2]) {
    /* Dynamic Look-Up Table Block: '<S12>/Interpolate BPOC'
     * Input0  Data Type:  Floating Point real32_T
     * Input1  Data Type:  Floating Point real32_T
     * Input2  Data Type:  Floating Point real32_T
     * Output0 Data Type:  Floating Point real32_T
     * Lookup Method: Linear_Endpoint
     *
     */
    LookUp_real32_T_real32_T( &(rtb_InterpolateBPOC_k), rtb_Switch1_i,
      LX2_B.Filter1_i.Switch, LX2_ConstP.pooled14, 10U, inst);
    rtb_SumofElements1 = rtb_InterpolateBPOC_k;
  } else {
    rtb_SumofElements1 = 0.0F;
  }

  /* End of Switch: '<S12>/Switch3' */

  /* Gain: '<S13>/mbar2bar' */
  rtb_Switch2_l = 0.001F * LX2_B.BusInput2.rPr_LX2_OffsetLimit;

  /* Logic: '<S13>/Logical Operator7' incorporates:
   *  Logic: '<S13>/Logical Operator8'
   *  Selector: '<S13>/Selector1'
   */
  rtb_LogicalOperator7_i = ((!rtb_LogicalOperator_f) && rtb_bSave_BPOC_enable[3]);

  /* Logic: '<S13>/Logical Operator2' incorporates:
   *  Logic: '<S13>/Logical Operator3'
   */
  rtb_RelationalOperator_b = ((!rtb_LogicalOperator7_i) || rtb_LogicalOperator_f);

  /* BusSelector: '<S6>/Bus Selector11' */
  for (i = 0; i < 5; i++) {
    rtb_rPr_LX2_offset_Lp_b[i] = LX2_B.BusInput.rP_Nom[i];
    rtb_rPr_LX2_offset_Lp_a[i] = LX2_B.BusInput.rP_Lp_b[i];
    rtb_rPr_LX2_offset_Lp_c[i] = LX2_B.BusInput.rP_Lp_a[i];
    rtb_rP_Lp_c[i] = LX2_B.BusInput.rP_Lp_c[i];
  }

  rtb_bLp_c_ena_n = LX2_B.BusInput.bLp_c_ena;

  /* End of BusSelector: '<S6>/Bus Selector11' */

  /* Logic: '<S13>/Logical Operator5' */
  rtb_LogicalOperator5_k = !rtb_LogicalOperator_f;

  /* Delay: '<S13>/Delay2' */
  didZcEventOccur = (((LX2_PrevZCSigState.Delay2_Reset_ZCE_k == LX2_POS_ZCSIG)
                      != rtb_RelationalOperator_b) &&
                     (LX2_PrevZCSigState.Delay2_Reset_ZCE_k !=
                      LX2_UNINITIALIZED_ZCSIG));
  LX2_PrevZCSigState.Delay2_Reset_ZCE_k = (uint8_T)rtb_RelationalOperator_b;
  if (rtb_RelationalOperator_b || didZcEventOccur) {
    LX2_DWork.icLoad_f = 1U;
  }

  for (i = 0; i < 11; i++) {
    if (LX2_DWork.icLoad_f != 0) {
      /* Switch: '<S13>/Switch5' incorporates:
       *  Constant: '<S13>/Constant5'
       */
      if (rtb_LogicalOperator5_k) {
        LX2_DWork.Delay2_DSTATE_d[i] = LX2_B.BusInput.rLX2_BPOC_Gas4[i];
      } else {
        LX2_DWork.Delay2_DSTATE_d[i] = 0.0F;
      }

      /* End of Switch: '<S13>/Switch5' */
    }

    rtb_Delay2_o1[i] = LX2_DWork.Delay2_DSTATE_d[i];
  }

  /* End of Delay: '<S13>/Delay2' */
  /* Dynamic Look-Up Table Block: '<S13>/Interpolate BPOC_actual'
   * Input0  Data Type:  Floating Point real32_T
   * Input1  Data Type:  Floating Point real32_T
   * Input2  Data Type:  Floating Point real32_T
   * Output0 Data Type:  Floating Point real32_T
   * Lookup Method: Linear_Endpoint
   *
   */
  LookUp_real32_T_real32_T( &(rtb_Divide), rtb_Delay2_o1, LX2_B.Filter1_i.Switch,
    LX2_ConstP.pooled14, 10U, inst);

  /* Sum: '<S13>/Sum1' incorporates:
   *  Product: '<S13>/Divide4'
   *  Selector: '<S13>/Selector2'
   *  Sum: '<S13>/Sum2'
   */
  rtb_Sum1_h = (rtb_UnitDelay2 - rtb_Divide) * rtb_splitfactor_Gas[3] +
    rtb_Divide;

  /* Logic: '<S13>/Logical Operator6' incorporates:
   *  Logic: '<S13>/Logical Operator4'
   */
  rtb_RelationalOperator_b = ((!rtb_LogicalOperator7_i) || rtb_LogicalOperator_f);

  /* Logic: '<S13>/Logical Operator1' */
  rtb_LogicalOperator5_k = !rtb_LogicalOperator_f;

  /* Delay: '<S13>/Delay1' */
  didZcEventOccur = (((LX2_PrevZCSigState.Delay1_Reset_ZCE_k == LX2_POS_ZCSIG)
                      != rtb_RelationalOperator_b) &&
                     (LX2_PrevZCSigState.Delay1_Reset_ZCE_k !=
                      LX2_UNINITIALIZED_ZCSIG));
  LX2_PrevZCSigState.Delay1_Reset_ZCE_k = (uint8_T)rtb_RelationalOperator_b;
  if (rtb_RelationalOperator_b || didZcEventOccur) {
    LX2_DWork.icLoad_c = 1U;
  }

  for (i = 0; i < 11; i++) {
    if (LX2_DWork.icLoad_c != 0) {
      /* Switch: '<S13>/Switch4' incorporates:
       *  Constant: '<S13>/Constant4'
       */
      if (rtb_LogicalOperator5_k) {
        LX2_DWork.Delay1_DSTATE_g[i] = LX2_B.BusInput.bLX2_BPOC_measured_Gas4[i];
      } else {
        LX2_DWork.Delay1_DSTATE_g[i] = FALSE;
      }

      /* End of Switch: '<S13>/Switch4' */
    }

    rtb_Delay1_c[i] = LX2_DWork.Delay1_DSTATE_g[i];
  }

  /* End of Delay: '<S13>/Delay1' */

  /* Selector: '<S13>/Selector6' incorporates:
   *  Constant: '<S6>/Constant8'
   */
  rtb_Divide = rtb_rPr_LX2_offset_Lp_a[4];

  /* Selector: '<S13>/Selector12' incorporates:
   *  Constant: '<S6>/Constant8'
   */
  rtb_Selector12 = rtb_rP_Lp_c[4];

  /* Switch: '<S28>/Switch' incorporates:
   *  Abs: '<S28>/Abs'
   *  Constant: '<S6>/Constant8'
   *  RelationalOperator: '<S28>/Relational Operator'
   *  Selector: '<S13>/Selector4'
   */
  if (2.22044605E-16F >= (real32_T)fabs(rtb_rPr_LX2_offset_Lp_b[4])) {
    rtb_UnitDelay3 = 2.22044605E-16F;
  } else {
    rtb_UnitDelay3 = rtb_rPr_LX2_offset_Lp_b[4];
  }

  /* End of Switch: '<S28>/Switch' */

  /* Gain: '<S13>/Gain1' incorporates:
   *  Constant: '<S6>/Constant8'
   *  Product: '<S13>/Divide'
   *  Selector: '<S13>/Selector5'
   */
  rtb_Lp2Lp3Lp_c_e[0] = rtb_Divide / rtb_UnitDelay3 * 100.0F;
  rtb_Lp2Lp3Lp_c_e[1] = rtb_rPr_LX2_offset_Lp_c[4] / rtb_UnitDelay3 * 100.0F;
  rtb_Lp2Lp3Lp_c_e[2] = rtb_Selector12 / rtb_UnitDelay3 * 100.0F;

  /* Gain: '<S13>/mbar2bar2' */
  rtb_mbar2bar2_m = 0.001F * rtb_Abs;

  /* Gain: '<S13>/mbar2bar3' */
  rtb_mbar2bar3_a = 0.001F * rtb_Switch2_b;

  /* BusSelector: '<S6>/Bus Selector12' */
  rtb_iWeight_Lp_0kW_k = LX2_B.BusInput1.iWeight_Lp_0kW;
  rtb_iWeight_Lp_b_e = LX2_B.BusInput1.iWeight_Lp_b;
  rtb_iWeight_Lp_a_h = LX2_B.BusInput1.iWeight_Lp_a;
  rtb_iWeight_Lp_c_e = LX2_B.BusInput1.iWeight_Lp_c;

  /* Gain: '<S13>/mbar2bar4' */
  rtb_mbar2bar4_g = 0.001F * LX2_B.BusInput2.rPr_LX2_OffsetLimit;

  /* MATLAB Function: '<S13>/Boost Pressure Offset Curve' */
  LX2_BoostPressureOffsetCurve(LX2_B.Filter1_i.Switch, rtb_Sum1_h, rtb_Delay2_o1,
    rtb_Delay1_c, rtb_Lp2Lp3Lp_c_e, rtb_bLp_c_ena_n, rtb_mbar2bar2_m,
    rtb_mbar2bar3_a, rtb_iWeight_Lp_0kW_k, rtb_iWeight_Lp_b_e,
    rtb_iWeight_Lp_a_h, rtb_iWeight_Lp_c_e, rtb_mbar2bar4_g,
    rtb_LogicalOperator7_i, &LX2_B.sf_BoostPressureOffsetCurve_a, inst);

  /* Gain: '<S13>/mbar2bar1' */
  rtb_SumofElements_o = 0.001F * rtb_LowerLimit_factor;
  for (i = 0; i < 11; i++) {
    /* Switch: '<S29>/Switch2' incorporates:
     *  RelationalOperator: '<S29>/LowerRelop1'
     *  RelationalOperator: '<S29>/UpperRelop'
     *  Switch: '<S29>/Switch'
     */
    if (LX2_B.sf_BoostPressureOffsetCurve_a.OUT_offset[i] > rtb_Switch2_l) {
      rtb_splitfactor_VISU_idx = rtb_Switch2_l;
    } else if (LX2_B.sf_BoostPressureOffsetCurve_a.OUT_offset[i] <
               rtb_SumofElements_o) {
      /* Switch: '<S29>/Switch' */
      rtb_splitfactor_VISU_idx = rtb_SumofElements_o;
    } else {
      rtb_splitfactor_VISU_idx =
        LX2_B.sf_BoostPressureOffsetCurve_a.OUT_offset[i];
    }

    /* Switch: '<S13>/Switch1' incorporates:
     *  Selector: '<S13>/Selector7'
     */
    if (rtb_Switch2_a_idx_2) {
      rtb_Switch1_it[i] = rtb_splitfactor_VISU_idx;
    } else {
      rtb_Switch1_it[i] = LX2_B.BusInput.rLX2_BPOC_Gas4[i];
    }

    /* End of Switch: '<S13>/Switch1' */

    /* Switch: '<S29>/Switch2' */
    rtb_Switch2_kq[i] = rtb_splitfactor_VISU_idx;
  }

  /* Switch: '<S13>/Switch3' incorporates:
   *  Constant: '<S13>/Constant2'
   *  Constant: '<S13>/Constant3'
   *  Selector: '<S13>/Selector3'
   */
  if (rtb_bBPOC_enable_a[3]) {
    /* Dynamic Look-Up Table Block: '<S13>/Interpolate BPOC'
     * Input0  Data Type:  Floating Point real32_T
     * Input1  Data Type:  Floating Point real32_T
     * Input2  Data Type:  Floating Point real32_T
     * Output0 Data Type:  Floating Point real32_T
     * Lookup Method: Linear_Endpoint
     *
     */
    LookUp_real32_T_real32_T( &(rtb_InterpolateBPOC), rtb_Switch1_it,
      LX2_B.Filter1_i.Switch, LX2_ConstP.pooled14, 10U, inst);
    rtb_SumofElements_o = rtb_InterpolateBPOC;
  } else {
    rtb_SumofElements_o = 0.0F;
  }

  /* End of Switch: '<S13>/Switch3' */

  /* Sum: '<S7>/Sum of Elements' incorporates:
   *  Product: '<S7>/Product'
   */
  rtb_SumofElements = ((rtb_Switch3 * rtb_splitfactor_Gas[0] +
                        rtb_SumofElements2 * rtb_splitfactor_Gas[1]) +
                       rtb_SumofElements1 * rtb_splitfactor_Gas[2]) +
    rtb_SumofElements_o * rtb_splitfactor_Gas[3];

  /* MATLAB Function: '<S7>/MATLAB Function' incorporates:
   *  Logic: '<S7>/Logical Operator1'
   *  Logic: '<S7>/Logical Operator2'
   *  Logic: '<S7>/Logical Operator6'
   *  MATLAB Function: '<S8>/MATLAB Function'
   *  SignalConversion: '<S38>/TmpSignal ConversionAt SFunction Inport4'
   *  UnitDelay: '<S7>/Unit Delay5'
   *  UnitDelay: '<S7>/Unit Delay6'
   */
  /* MATLAB Function 'Leanox 2.0/Controller/MATLAB Function': '<S38>:1' */
  if (rtb_Compare_n || rtb_LogicalOperator6_a || (!bCtrl_enable)) {
    /* '<S38>:1:9' */
    /* '<S38>:1:10' */
    rtb_Reset = TRUE;

    /* '<S38>:1:11' */
    b_y = 0.0F;
  } else if (rtb_UnitDelay1) {
    /* '<S38>:1:12' */
    /* '<S38>:1:13' */
    rtb_Reset = TRUE;

    /* '<S38>:1:14' */
    b_y = LX2_DWork.UnitDelay6_DSTATE;
  } else if (rtb_Switch2_a_idx || rtb_Switch2_a_idx_0 || rtb_Switch2_a_idx_1 ||
             rtb_Switch2_a_idx_2) {
    /* '<S38>:1:15' */
    /* '<S38>:1:16' */
    rtb_Reset = TRUE;

    /* '<S38>:1:17' */
    b_y = (LX2_DWork.UnitDelay5_DSTATE - rtb_SumofElements) +
      LX2_DWork.UnitDelay6_DSTATE;
  } else {
    /* '<S38>:1:19' */
    rtb_Reset = FALSE;

    /* '<S38>:1:20' */
    b_y = LX2_DWork.y0_1;
  }

  /* '<S38>:1:22' */
  LX2_DWork.y0_1 = b_y;

  /* DiscreteIntegrator: '<S36>/Discrete-Time Integrator' incorporates:
   *  MATLAB Function: '<S7>/MATLAB Function'
   */
  if (LX2_DWork.DiscreteTimeIntegrator_IC_LOADI != 0) {
    LX2_DWork.DiscreteTimeIntegrator_DSTATE = b_y;
  }

  if (rtb_Reset || (LX2_DWork.DiscreteTimeIntegrator_PrevRese != 0)) {
    LX2_DWork.DiscreteTimeIntegrator_DSTATE = b_y;
  }

  rtb_DiscreteTimeIntegrator = LX2_DWork.DiscreteTimeIntegrator_DSTATE;

  /* Sum: '<S7>/Sum2' incorporates:
   *  DiscreteIntegrator: '<S36>/Discrete-Time Integrator'
   */
  rtb_Sum2_e = LX2_DWork.DiscreteTimeIntegrator_DSTATE + rtb_SumofElements;

  /* Switch: '<S7>/Switch6' incorporates:
   *  Gain: '<S7>/mbar2bar'
   *  MATLAB Function: '<S8>/MATLAB Function'
   *  UnitDelay: '<S7>/Unit Delay4'
   */
  if (b_bEng_knock) {
    rtb_Switch6 = LX2_DWork.UnitDelay4_DSTATE;
  } else {
    rtb_Switch6 = 0.001F * rtb_LowerLimit_factor;
  }

  /* End of Switch: '<S7>/Switch6' */

  /* Switch: '<S39>/Switch2' incorporates:
   *  RelationalOperator: '<S39>/LowerRelop1'
   *  RelationalOperator: '<S39>/UpperRelop'
   *  Switch: '<S39>/Switch'
   */
  if (rtb_Sum2_e > rtb_Switch7) {
    rtb_UnitDelay3 = rtb_Switch7;
  } else if (rtb_Sum2_e < rtb_Switch6) {
    /* Switch: '<S39>/Switch' */
    rtb_UnitDelay3 = rtb_Switch6;
  } else {
    rtb_UnitDelay3 = rtb_Sum2_e;
  }

  /* End of Switch: '<S39>/Switch2' */

  /* Logic: '<S52>/Logical Operator2' */
  rtb_Compare_n = (LX2_B.BusInput.bLeanox_Adjust && LX2_B.BusInput2.bLX2_enable);

  /* Delay: '<S41>/Delay' */
  didZcEventOccur = (((LX2_PrevZCSigState.Delay_Reset_ZCE == LX2_POS_ZCSIG) !=
                      rtb_Compare_n) && (LX2_PrevZCSigState.Delay_Reset_ZCE !=
    LX2_UNINITIALIZED_ZCSIG));
  LX2_PrevZCSigState.Delay_Reset_ZCE = (uint8_T)rtb_Compare_n;
  if (rtb_Compare_n || didZcEventOccur) {
    LX2_DWork.icLoad_i = 1U;
  }

  if (LX2_DWork.icLoad_i != 0) {
    LX2_DWork.Delay_DSTATE = rtb_UnitDelay3;
  }

  rtb_Switch2_l = LX2_DWork.Delay_DSTATE;

  /* End of Delay: '<S41>/Delay' */

  /* Sum: '<S41>/Difference Inputs1' incorporates:
   *  Switch: '<S41>/etaVolConst'
   */
  rtb_UnitDelay2 = rtb_UnitDelay3 - rtb_Switch2_l;

  /* Switch: '<S49>/Switch2' incorporates:
   *  RelationalOperator: '<S49>/LowerRelop1'
   */
  if (!(rtb_UnitDelay2 > rtb_Switch2_kt)) {
    /* Product: '<S41>/delta fall limit' incorporates:
     *  UnaryMinus: '<S7>/Unary Minus1'
     */
    rtb_UnitDelay3 = -rtb_Gain3 * 0.1F;

    /* Switch: '<S49>/Switch' incorporates:
     *  RelationalOperator: '<S49>/UpperRelop'
     */
    if (rtb_UnitDelay2 < rtb_UnitDelay3) {
      rtb_Switch2_kt = rtb_UnitDelay3;
    } else {
      rtb_Switch2_kt = rtb_UnitDelay2;
    }

    /* End of Switch: '<S49>/Switch' */
  }

  /* End of Switch: '<S49>/Switch2' */

  /* Sum: '<S41>/Difference Inputs2' */
  rtb_Switch2_kt += rtb_Switch2_l;

  /* SignalConversion: '<S5>/TmpSignal ConversionAtBus CreatorInport2' incorporates:
   *  Constant: '<S5>/Constant'
   */
  rtb_bLX2_save[0] = FALSE;
  rtb_bLX2_save[1] = rtb_Switch2_a_idx;
  rtb_bLX2_save[2] = rtb_Switch2_a_idx_0;
  rtb_bLX2_save[3] = rtb_Switch2_a_idx_1;
  rtb_bLX2_save[4] = rtb_Switch2_a_idx_2;

  /* Dynamic Look-Up Table Block: '<S10>/Interpolate BPOC at Lp2 (half load)'
   * Input0  Data Type:  Floating Point real32_T
   * Input1  Data Type:  Floating Point real32_T
   * Input2  Data Type:  Floating Point real32_T
   * Output0 Data Type:  Floating Point real32_T
   * Lookup Method: Linear_Endpoint
   *
   */
  LookUp_real32_T_real32_T( &(rtb_Switch2_l), rtb_Switch1, rtb_Lp2Lp3Lp_c[0],
    LX2_ConstP.pooled14, 10U, inst);

  /* Dynamic Look-Up Table Block: '<S11>/Interpolate BPOC at Lp2 (half load)'
   * Input0  Data Type:  Floating Point real32_T
   * Input1  Data Type:  Floating Point real32_T
   * Input2  Data Type:  Floating Point real32_T
   * Output0 Data Type:  Floating Point real32_T
   * Lookup Method: Linear_Endpoint
   *
   */
  LookUp_real32_T_real32_T( &(rtb_Divide), rtb_Switch1_m, rtb_Lp2Lp3Lp_c_n[0],
    LX2_ConstP.pooled14, 10U, inst);

  /* Dynamic Look-Up Table Block: '<S12>/Interpolate BPOC at Lp2 (half load)'
   * Input0  Data Type:  Floating Point real32_T
   * Input1  Data Type:  Floating Point real32_T
   * Input2  Data Type:  Floating Point real32_T
   * Output0 Data Type:  Floating Point real32_T
   * Lookup Method: Linear_Endpoint
   *
   */
  LookUp_real32_T_real32_T( &(rtb_Abs), rtb_Switch1_i, rtb_Lp2Lp3Lp_c_l[0],
    LX2_ConstP.pooled14, 10U, inst);

  /* Dynamic Look-Up Table Block: '<S13>/Interpolate BPOC at Lp2 (half load)'
   * Input0  Data Type:  Floating Point real32_T
   * Input1  Data Type:  Floating Point real32_T
   * Input2  Data Type:  Floating Point real32_T
   * Output0 Data Type:  Floating Point real32_T
   * Lookup Method: Linear_Endpoint
   *
   */
  LookUp_real32_T_real32_T( &(rtb_Switch2_b), rtb_Switch1_it, rtb_Lp2Lp3Lp_c_e[0],
    LX2_ConstP.pooled14, 10U, inst);

  /* SignalConversion: '<S5>/TmpSignal ConversionAtBus CreatorInport3' incorporates:
   *  Constant: '<S5>/Constant1'
   */
  rtb_rPr_LX2_offset_Lp_b[0] = 0.0F;
  rtb_rPr_LX2_offset_Lp_b[1] = rtb_Switch2_l;
  rtb_rPr_LX2_offset_Lp_b[2] = rtb_Divide;
  rtb_rPr_LX2_offset_Lp_b[3] = rtb_Abs;
  rtb_rPr_LX2_offset_Lp_b[4] = rtb_Switch2_b;

  /* Dynamic Look-Up Table Block: '<S10>/Interpolate BPOC at Lp3 (full load)'
   * Input0  Data Type:  Floating Point real32_T
   * Input1  Data Type:  Floating Point real32_T
   * Input2  Data Type:  Floating Point real32_T
   * Output0 Data Type:  Floating Point real32_T
   * Lookup Method: Linear_Endpoint
   *
   */
  LookUp_real32_T_real32_T( &(rtb_Switch2_l), rtb_Switch1, rtb_Lp2Lp3Lp_c[1],
    LX2_ConstP.pooled14, 10U, inst);

  /* Dynamic Look-Up Table Block: '<S11>/Interpolate BPOC at Lp3 (full load)'
   * Input0  Data Type:  Floating Point real32_T
   * Input1  Data Type:  Floating Point real32_T
   * Input2  Data Type:  Floating Point real32_T
   * Output0 Data Type:  Floating Point real32_T
   * Lookup Method: Linear_Endpoint
   *
   */
  LookUp_real32_T_real32_T( &(rtb_Divide), rtb_Switch1_m, rtb_Lp2Lp3Lp_c_n[1],
    LX2_ConstP.pooled14, 10U, inst);

  /* Dynamic Look-Up Table Block: '<S12>/Interpolate BPOC at Lp3 (full load)'
   * Input0  Data Type:  Floating Point real32_T
   * Input1  Data Type:  Floating Point real32_T
   * Input2  Data Type:  Floating Point real32_T
   * Output0 Data Type:  Floating Point real32_T
   * Lookup Method: Linear_Endpoint
   *
   */
  LookUp_real32_T_real32_T( &(rtb_Abs), rtb_Switch1_i, rtb_Lp2Lp3Lp_c_l[1],
    LX2_ConstP.pooled14, 10U, inst);

  /* Dynamic Look-Up Table Block: '<S13>/Interpolate BPOC at Lp3 (full load)'
   * Input0  Data Type:  Floating Point real32_T
   * Input1  Data Type:  Floating Point real32_T
   * Input2  Data Type:  Floating Point real32_T
   * Output0 Data Type:  Floating Point real32_T
   * Lookup Method: Linear_Endpoint
   *
   */
  LookUp_real32_T_real32_T( &(rtb_Switch2_b), rtb_Switch1_it, rtb_Lp2Lp3Lp_c_e[1],
    LX2_ConstP.pooled14, 10U, inst);

  /* SignalConversion: '<S5>/TmpSignal ConversionAtBus CreatorInport4' incorporates:
   *  Constant: '<S5>/Constant2'
   */
  rtb_rPr_LX2_offset_Lp_a[0] = 0.0F;
  rtb_rPr_LX2_offset_Lp_a[1] = rtb_Switch2_l;
  rtb_rPr_LX2_offset_Lp_a[2] = rtb_Divide;
  rtb_rPr_LX2_offset_Lp_a[3] = rtb_Abs;
  rtb_rPr_LX2_offset_Lp_a[4] = rtb_Switch2_b;

  /* Switch: '<S10>/Switch2' incorporates:
   *  Constant: '<S10>/Constant1'
   *  Constant: '<S10>/Constant2'
   */
  if (rtb_bLp_c_ena) {
    /* Dynamic Look-Up Table Block: '<S10>/Interpolate BPOC at Lp_c (25% load)'
     * Input0  Data Type:  Floating Point real32_T
     * Input1  Data Type:  Floating Point real32_T
     * Input2  Data Type:  Floating Point real32_T
     * Output0 Data Type:  Floating Point real32_T
     * Lookup Method: Linear_Endpoint
     *
     */
    LookUp_real32_T_real32_T( &(rtb_InterpolateBPOCatLp_c25lo_e), rtb_Switch1,
      rtb_Lp2Lp3Lp_c[2], LX2_ConstP.pooled14, 10U, inst);
    rtb_Switch2_l = rtb_InterpolateBPOCatLp_c25lo_e;
  } else {
    rtb_Switch2_l = 0.0F;
  }

  /* End of Switch: '<S10>/Switch2' */

  /* Switch: '<S11>/Switch2' incorporates:
   *  Constant: '<S11>/Constant1'
   *  Constant: '<S11>/Constant2'
   */
  if (rtb_bLp_c_ena_i) {
    /* Dynamic Look-Up Table Block: '<S11>/Interpolate BPOC at Lp_c (25% load)'
     * Input0  Data Type:  Floating Point real32_T
     * Input1  Data Type:  Floating Point real32_T
     * Input2  Data Type:  Floating Point real32_T
     * Output0 Data Type:  Floating Point real32_T
     * Lookup Method: Linear_Endpoint
     *
     */
    LookUp_real32_T_real32_T( &(rtb_InterpolateBPOCatLp_c25lo_l), rtb_Switch1_m,
      rtb_Lp2Lp3Lp_c_n[2], LX2_ConstP.pooled14, 10U, inst);
    rtb_Divide = rtb_InterpolateBPOCatLp_c25lo_l;
  } else {
    rtb_Divide = 0.0F;
  }

  /* End of Switch: '<S11>/Switch2' */

  /* Switch: '<S12>/Switch2' incorporates:
   *  Constant: '<S12>/Constant1'
   *  Constant: '<S12>/Constant2'
   */
  if (rtb_bLp_c_ena_h) {
    /* Dynamic Look-Up Table Block: '<S12>/Interpolate BPOC at Lp_c (25% load)'
     * Input0  Data Type:  Floating Point real32_T
     * Input1  Data Type:  Floating Point real32_T
     * Input2  Data Type:  Floating Point real32_T
     * Output0 Data Type:  Floating Point real32_T
     * Lookup Method: Linear_Endpoint
     *
     */
    LookUp_real32_T_real32_T( &(rtb_InterpolateBPOCatLp_c25lo_h), rtb_Switch1_i,
      rtb_Lp2Lp3Lp_c_l[2], LX2_ConstP.pooled14, 10U, inst);
    rtb_Abs = rtb_InterpolateBPOCatLp_c25lo_h;
  } else {
    rtb_Abs = 0.0F;
  }

  /* End of Switch: '<S12>/Switch2' */

  /* Switch: '<S13>/Switch2' incorporates:
   *  Constant: '<S13>/Constant1'
   *  Constant: '<S13>/Constant2'
   */
  if (rtb_bLp_c_ena_n) {
    /* Dynamic Look-Up Table Block: '<S13>/Interpolate BPOC at Lp_c (25% load)'
     * Input0  Data Type:  Floating Point real32_T
     * Input1  Data Type:  Floating Point real32_T
     * Input2  Data Type:  Floating Point real32_T
     * Output0 Data Type:  Floating Point real32_T
     * Lookup Method: Linear_Endpoint
     *
     */
    LookUp_real32_T_real32_T( &(rtb_InterpolateBPOCatLp_c25load), rtb_Switch1_it,
      rtb_Lp2Lp3Lp_c_e[2], LX2_ConstP.pooled14, 10U, inst);
    rtb_Switch2_b = rtb_InterpolateBPOCatLp_c25load;
  } else {
    rtb_Switch2_b = 0.0F;
  }

  /* End of Switch: '<S13>/Switch2' */

  /* SignalConversion: '<S5>/TmpSignal ConversionAtBus CreatorInport5' incorporates:
   *  Constant: '<S5>/Constant3'
   */
  rtb_rPr_LX2_offset_Lp_c[0] = 0.0F;
  rtb_rPr_LX2_offset_Lp_c[1] = rtb_Switch2_l;
  rtb_rPr_LX2_offset_Lp_c[2] = rtb_Divide;
  rtb_rPr_LX2_offset_Lp_c[3] = rtb_Abs;
  rtb_rPr_LX2_offset_Lp_c[4] = rtb_Switch2_b;

  /* MATLAB Function: '<S14>/MATLAB Function' */
  /* MATLAB Function 'Leanox 2.0/BPOC/Visu/MATLAB Function': '<S31>:1' */
  /* persistent y0_1 */
  /*   */
  /*  if isempty(y0_1) */
  /*      y0_1 = single(0); */
  /*  end */
  /*  define output vector */
  /* '<S31>:1:11' */
  if (!LX2_B.BusInput2.bLX2_enable) {
    /* '<S31>:1:13' */
    /* '<S31>:1:14' */
    rtb_UnitDelay3 = 0.0F;

    /* '<S31>:1:15' */
    rtb_UnitDelay2 = 0.0F;

    /* '<S31>:1:16' */
    rtb_Gain3 = 0.0F;

    /* '<S31>:1:17' */
    rtb_splitfactor_VISU_idx = 0.0F;
  } else if (LX2_B.BusInput2.bLX2_enable && LX2_B.BusInput.bLX2_active) {
    /* '<S31>:1:19' */
    /* '<S31>:1:20' */
    rtb_UnitDelay3 = rtb_splitfactor_Gas[0];
    rtb_UnitDelay2 = rtb_splitfactor_Gas[1];
    rtb_Gain3 = rtb_splitfactor_Gas[2];
    rtb_splitfactor_VISU_idx = rtb_splitfactor_Gas[3];
  } else {
    /*  (bLX2_enable == true) && (bLX2_active == false) */
    if (LX2_B.BusInput.iIdx_Gtyp_Dem < 4) {
      /* '<S31>:1:23' */
      /* '<S31>:1:24' */
      rtb_UnitDelay3 = (1.0F - LX2_B.BusInput.rGT_QualMix_1_2) * (1.0F -
        LX2_B.BusInput.rGT_RatioMix);

      /* '<S31>:1:25' */
      rtb_UnitDelay2 = (1.0F - LX2_B.BusInput.rGT_RatioMix) *
        LX2_B.BusInput.rGT_QualMix_1_2;

      /* '<S31>:1:26' */
      rtb_Gain3 = LX2_B.BusInput.rGT_RatioMix;

      /* '<S31>:1:27' */
      rtb_splitfactor_VISU_idx = 0.0F;
    } else if (LX2_B.BusInput.iIdx_Gtyp_Dem == 4) {
      /* '<S31>:1:29' */
      /* '<S31>:1:30' */
      rtb_UnitDelay3 = 0.0F;

      /* '<S31>:1:31' */
      rtb_UnitDelay2 = 0.0F;

      /* '<S31>:1:32' */
      rtb_Gain3 = 0.0F;

      /* '<S31>:1:33' */
      rtb_splitfactor_VISU_idx = 1.0F;
    } else {
      /*  undefined Gastype */
      /* '<S31>:1:36' */
      rtb_UnitDelay3 = 0.0F;

      /* '<S31>:1:37' */
      rtb_UnitDelay2 = 0.0F;

      /* '<S31>:1:38' */
      rtb_Gain3 = 0.0F;

      /* '<S31>:1:39' */
      rtb_splitfactor_VISU_idx = 0.0F;
    }
  }

  /* End of MATLAB Function: '<S14>/MATLAB Function' */

  /* Selector: '<S14>/Selector9' */
  /*  y0_1 = y0; */
  rtb_Switch2_l = rtb_UnitDelay3;

  /* Product: '<S14>/Product4' */
  for (i = 0; i < 11; i++) {
    /* Switch: '<S14>/Switch10' incorporates:
     *  Constant: '<S14>/Constant18'
     */
    if (rtb_Switch2_l != 0.0F) {
      tmp_1 = LX2_B.BusInput.rLX2_BPOC_Gas1[i];
    } else {
      tmp_1 = 0.0F;
    }

    /* End of Switch: '<S14>/Switch10' */
    rtb_Product4[i] = rtb_Switch2_l * tmp_1;
  }

  /* End of Product: '<S14>/Product4' */

  /* Selector: '<S14>/Selector10' */
  rtb_Switch2_l = rtb_UnitDelay2;

  /* Product: '<S14>/Product5' */
  for (i = 0; i < 11; i++) {
    /* Switch: '<S14>/Switch8' incorporates:
     *  Constant: '<S14>/Constant19'
     */
    if (rtb_Switch2_l != 0.0F) {
      tmp_1 = LX2_B.BusInput.rLX2_BPOC_Gas2[i];
    } else {
      tmp_1 = 0.0F;
    }

    /* End of Switch: '<S14>/Switch8' */
    rtb_Product5[i] = rtb_Switch2_l * tmp_1;
  }

  /* End of Product: '<S14>/Product5' */

  /* Selector: '<S14>/Selector11' */
  rtb_Switch2_l = rtb_Gain3;

  /* Product: '<S14>/Product6' */
  for (i = 0; i < 11; i++) {
    /* Switch: '<S14>/Switch9' incorporates:
     *  Constant: '<S14>/Constant21'
     */
    if (rtb_Switch2_l != 0.0F) {
      tmp_1 = LX2_B.BusInput.rLX2_BPOC_Gas3[i];
    } else {
      tmp_1 = 0.0F;
    }

    /* End of Switch: '<S14>/Switch9' */
    rtb_Product6[i] = rtb_Switch2_l * tmp_1;
  }

  /* End of Product: '<S14>/Product6' */

  /* Selector: '<S14>/Selector12' */
  rtb_Switch2_l = rtb_splitfactor_VISU_idx;
  for (i = 0; i < 11; i++) {
    /* Switch: '<S14>/Switch11' incorporates:
     *  Constant: '<S14>/Constant23'
     */
    if (rtb_Switch2_l != 0.0F) {
      tmp_1 = LX2_B.BusInput.rLX2_BPOC_Gas4[i];
    } else {
      tmp_1 = 0.0F;
    }

    /* End of Switch: '<S14>/Switch11' */

    /* Product: '<S14>/Product7' */
    rtb_Product7[i] = rtb_Switch2_l * tmp_1;

    /* Switch: '<S14>/Switch6' incorporates:
     *  Constant: '<S14>/Constant7'
     *  Selector: '<S14>/Selector5'
     */
    if (rtb_UnitDelay3 != 0.0F) {
      rtb_Switch5_kl[i] = (int8_T)LX2_B.BusInput.bLX2_BPOC_measured_Gas1[i];
    } else {
      rtb_Switch5_kl[i] = 0;
    }

    /* End of Switch: '<S14>/Switch6' */

    /* Switch: '<S14>/Switch4' incorporates:
     *  Constant: '<S14>/Constant10'
     *  Selector: '<S14>/Selector6'
     */
    if (rtb_UnitDelay2 != 0.0F) {
      rtb_Switch4[i] = (int8_T)LX2_B.BusInput.bLX2_BPOC_measured_Gas2[i];
    } else {
      rtb_Switch4[i] = 0;
    }

    /* End of Switch: '<S14>/Switch4' */

    /* Switch: '<S14>/Switch5' incorporates:
     *  Constant: '<S14>/Constant11'
     *  Selector: '<S14>/Selector7'
     */
    if (rtb_Gain3 != 0.0F) {
      rtb_Switch6_j[i] = (int8_T)LX2_B.BusInput.bLX2_BPOC_measured_Gas3[i];
    } else {
      rtb_Switch6_j[i] = 0;
    }

    /* End of Switch: '<S14>/Switch5' */

    /* Switch: '<S14>/Switch7' incorporates:
     *  Constant: '<S14>/Constant13'
     *  Selector: '<S14>/Selector8'
     */
    if (rtb_splitfactor_VISU_idx != 0.0F) {
      rtb_rLX2_BPOC[i] = (int8_T)LX2_B.BusInput.bLX2_BPOC_measured_Gas4[i];
    } else {
      rtb_rLX2_BPOC[i] = 0;
    }

    /* End of Switch: '<S14>/Switch7' */
  }

  /* Logic: '<S37>/Logical Operator4' incorporates:
   *  Bias: '<S37>/Bias'
   *  Bias: '<S37>/Bias1'
   *  Gain: '<S37>/mbar2bar'
   *  Gain: '<S37>/mbar2bar1'
   *  RelationalOperator: '<S37>/Relational Operator2'
   *  RelationalOperator: '<S37>/Relational Operator3'
   */
  rtb_LogicalOperator4_g = ((rtb_Switch2_kt >= 0.001F *
    LX2_B.BusInput2.rPr_LX2_OffsetLimit + -1.1920929E-5F) || (rtb_Switch2_kt <=
    0.001F * rtb_LowerLimit_factor + 1.1920929E-5F));

  /* Outputs for Atomic SubSystem: '<S37>/TON' */
  LX2_TON(rtb_LogicalOperator4_g, rtb_rLX2_inLimitSetup_Time, &LX2_B.TON_b,
          &LX2_DWork.TON_b, inst);

  /* End of Outputs for SubSystem: '<S37>/TON' */

  /* BusCreator: '<S5>/Bus Creator' incorporates:
   *  Logic: '<S14>/Logical Operator'
   *  Logic: '<S14>/Logical Operator1'
   *  Logic: '<S14>/Logical Operator2'
   *  Sum: '<S14>/Add'
   */
  LX2_Y.tLX2_OUT_c.rPr_LX2_offset = rtb_Switch2_kt;
  for (i = 0; i < 5; i++) {
    LX2_Y.tLX2_OUT_c.bLX2_save[i] = rtb_bLX2_save[i];
    LX2_Y.tLX2_OUT_c.rPr_LX2_offset_Lp_b[i] = rtb_rPr_LX2_offset_Lp_b[i];
    LX2_Y.tLX2_OUT_c.rPr_LX2_offset_Lp_a[i] = rtb_rPr_LX2_offset_Lp_a[i];
    LX2_Y.tLX2_OUT_c.rPr_LX2_offset_Lp_c[i] = rtb_rPr_LX2_offset_Lp_c[i];
  }

  for (i = 0; i < 11; i++) {
    LX2_Y.tLX2_OUT_c.rLX2_BPOC_Gas1[i] = rtb_Switch2[i];
    LX2_Y.tLX2_OUT_c.bLX2_BPOC_measured_Gas1[i] =
      LX2_B.sf_BoostPressureOffsetCurve.OUT_measured[i];
    LX2_Y.tLX2_OUT_c.rLX2_BPOC_Gas2[i] = rtb_Switch2_j[i];
    LX2_Y.tLX2_OUT_c.bLX2_BPOC_measured_Gas2[i] =
      LX2_B.sf_BoostPressureOffsetCurve_f.OUT_measured[i];
    LX2_Y.tLX2_OUT_c.rLX2_BPOC_Gas3[i] = rtb_Switch2_k[i];
    LX2_Y.tLX2_OUT_c.bLX2_BPOC_measured_Gas3[i] =
      LX2_B.sf_BoostPressureOffsetCurve_d.OUT_measured[i];
    LX2_Y.tLX2_OUT_c.rLX2_BPOC_Gas4[i] = rtb_Switch2_kq[i];
    LX2_Y.tLX2_OUT_c.bLX2_BPOC_measured_Gas4[i] =
      LX2_B.sf_BoostPressureOffsetCurve_a.OUT_measured[i];
    LX2_Y.tLX2_OUT_c.rLX2_BPOC[i] = ((rtb_Product4[i] + rtb_Product5[i]) +
      rtb_Product6[i]) + rtb_Product7[i];
    LX2_Y.tLX2_OUT_c.bLX2_BPOC_measured[i] = ((rtb_Switch5_kl[i] != 0) ||
      (rtb_Switch4[i] != 0) || (rtb_Switch6_j[i] != 0) || (rtb_rLX2_BPOC[i] != 0));
  }

  LX2_Y.tLX2_OUT_c.bBPOC_enable = (rtb_bBPOC_enable_a[0] || rtb_bBPOC_enable_a[1]
    || rtb_bBPOC_enable_a[2] || rtb_bBPOC_enable_a[3]);
  LX2_Y.tLX2_OUT_c.bBPOC_save_enable = (rtb_bSave_BPOC_enable[0] ||
    rtb_bSave_BPOC_enable[1] || rtb_bSave_BPOC_enable[2] ||
    rtb_bSave_BPOC_enable[3]);
  LX2_Y.tLX2_OUT_c.bLX2_inLimit = LX2_B.TON_b.LogicalOperator3;

  /* End of BusCreator: '<S5>/Bus Creator' */

  /* BusCreator: '<S8>/Bus Creator' */
  rtb_LogicalOperator5_k = rtb_LogicalOperator_f;

  /* Switch: '<S7>/Switch2' incorporates:
   *  RelationalOperator: '<S34>/FixPt Relational Operator'
   *  Sum: '<S7>/Sum9'
   *  UnitDelay: '<S34>/Delay Input1'
   */
  if ((uint8_T)((int32_T)LX2_B.BusInput.bNOx_valid - ((int32_T)
        LX2_B.BusInput.bNOx_valid > (int32_T)LX2_DWork.DelayInput1_DSTATE)) != 0)
  {
    /* Saturate: '<S7>/Saturation' */
    if (rtb_rNOx_act_g >= 300.0F) {
      rtb_UnitDelay3 = 300.0F;
    } else if (rtb_rNOx_act_g <= 20.0F) {
      rtb_UnitDelay3 = 20.0F;
    } else {
      rtb_UnitDelay3 = rtb_rNOx_act_g;
    }

    /* End of Saturate: '<S7>/Saturation' */
  } else {
    rtb_UnitDelay3 = LX2_B.BusInput.rNOx_set;
  }

  /* End of Switch: '<S7>/Switch2' */

  /* Outputs for Atomic SubSystem: '<S7>/Filter' */
  /* RelationalOperator: '<S35>/Relational Operator' incorporates:
   *  Constant: '<S35>/Constant'
   */
  rtb_RelationalOperator_b = (LX2_B.BusInput2.rFilterConst_NOx > 0.0F);

  /* Logic: '<S35>/Logical Operator' incorporates:
   *  Logic: '<S35>/Logical Operator1'
   *  Logic: '<S7>/Logical Operator3'
   *  Logic: '<S7>/Logical Operator4'
   */
  rtb_LogicalOperator_d = ((!LX2_B.BusInput.bNOx_valid) ||
    rtb_LogicalOperator6_a || (!rtb_RelationalOperator_b));

  /* DiscreteIntegrator: '<S35>/Discrete-Time Integrator' */
  if (LX2_DWork.DiscreteTimeIntegrator_IC_LOA_l != 0) {
    LX2_DWork.DiscreteTimeIntegrator_DSTATE_n = rtb_UnitDelay3;
  }

  if (rtb_LogicalOperator_d || (LX2_DWork.DiscreteTimeIntegrator_PrevRe_a != 0))
  {
    LX2_DWork.DiscreteTimeIntegrator_DSTATE_n = rtb_UnitDelay3;
  }

  /* Switch: '<S35>/Switch' incorporates:
   *  DiscreteIntegrator: '<S35>/Discrete-Time Integrator'
   */
  if (rtb_RelationalOperator_b) {
    rtb_splitfactor_VISU_idx = LX2_DWork.DiscreteTimeIntegrator_DSTATE_n;
  } else {
    rtb_splitfactor_VISU_idx = rtb_rNOx_act_g;
  }

  /* End of Switch: '<S35>/Switch' */

  /* Update for DiscreteIntegrator: '<S35>/Discrete-Time Integrator' */
  LX2_DWork.DiscreteTimeIntegrator_IC_LOA_l = 0U;

  /* Switch: '<S42>/Switch' incorporates:
   *  Abs: '<S42>/Abs'
   *  Constant: '<S42>/Constant2'
   *  RelationalOperator: '<S42>/Relational Operator'
   */
  if (0.1F >= (real32_T)fabs(LX2_B.BusInput2.rFilterConst_NOx)) {
    tmp_1 = 0.1F;
  } else {
    tmp_1 = LX2_B.BusInput2.rFilterConst_NOx;
  }

  /* End of Switch: '<S42>/Switch' */

  /* Update for DiscreteIntegrator: '<S35>/Discrete-Time Integrator' incorporates:
   *  DiscreteIntegrator: '<S35>/Discrete-Time Integrator'
   *  Product: '<S35>/Divide4'
   *  Sum: '<S35>/Sum4'
   */
  LX2_DWork.DiscreteTimeIntegrator_DSTATE_n += (rtb_rNOx_act_g -
    LX2_DWork.DiscreteTimeIntegrator_DSTATE_n) / tmp_1 * 0.1F;
  if (rtb_LogicalOperator_d) {
    LX2_DWork.DiscreteTimeIntegrator_PrevRe_a = 1;
  } else {
    LX2_DWork.DiscreteTimeIntegrator_PrevRe_a = 0;
  }

  /* End of Outputs for SubSystem: '<S7>/Filter' */

  /* Sum: '<S7>/Sum' */
  rtb_UnitDelay3 = rtb_splitfactor_VISU_idx - LX2_B.BusInput.rNOx_set;

  /* Switch: '<S40>/Switch2' incorporates:
   *  Gain: '<S7>/LowerLim_factor'
   *  RelationalOperator: '<S40>/LowerRelop1'
   *  RelationalOperator: '<S40>/UpperRelop'
   *  Switch: '<S40>/Switch'
   */
  if (rtb_UnitDelay3 > LX2_B.BusInput1.rCtrlError_Limit) {
    rtb_Switch2_l = LX2_B.BusInput1.rCtrlError_Limit;
  } else if (rtb_UnitDelay3 < -LX2_B.BusInput1.rCtrlError_Limit) {
    /* Switch: '<S40>/Switch' incorporates:
     *  Gain: '<S7>/LowerLim_factor'
     */
    rtb_Switch2_l = -LX2_B.BusInput1.rCtrlError_Limit;
  } else {
    /* Switch: '<S40>/Switch' */
    rtb_Switch2_l = rtb_UnitDelay3;
  }

  /* End of Switch: '<S40>/Switch2' */

  /* Switch: '<S7>/Switch1' incorporates:
   *  Constant: '<S33>/Constant'
   *  Constant: '<S7>/Constant'
   *  Logic: '<S7>/Logical Operator5'
   *  MATLAB Function: '<S8>/MATLAB Function'
   *  RelationalOperator: '<S33>/Compare'
   */
  if ((rtb_Switch7 <= 0.0F) || bCtrl_freeze) {
    rtb_Divide = 0.0F;
  } else {
    rtb_Divide = rtb_Switch2_l;
  }

  /* End of Switch: '<S7>/Switch1' */

  /* Abs: '<S45>/Abs' */
  rtb_Abs = (real32_T)fabs(rtb_Switch_nq);

  /* Switch: '<S45>/Switch' incorporates:
   *  Constant: '<S45>/Constant2'
   *  RelationalOperator: '<S45>/Relational Operator'
   */
  if (0.1F >= rtb_Abs) {
    rtb_Switch_nq = 0.1F;
  }

  /* End of Switch: '<S45>/Switch' */

  /* Product: '<S36>/Divide' */
  rtb_Divide /= rtb_Switch_nq;

  /* Signum: '<S44>/Sign2' incorporates:
   *  DataTypeConversion: '<S44>/Data Type Conversion2'
   */
  if (rtb_Sum2_e < 0.0F) {
    rtb_Sum2_e_0 = -1.0;
  } else if (rtb_Sum2_e > 0.0F) {
    rtb_Sum2_e_0 = 1.0;
  } else {
    rtb_Sum2_e_0 = rtb_Sum2_e;
  }

  /* Signum: '<S44>/Sign1' incorporates:
   *  DataTypeConversion: '<S44>/Data Type Conversion3'
   */
  if (rtb_Divide < 0.0F) {
    tmp_2 = -1.0;
  } else if (rtb_Divide > 0.0F) {
    tmp_2 = 1.0;
  } else {
    tmp_2 = rtb_Divide;
  }

  /* Logic: '<S44>/Logical Operator' incorporates:
   *  Logic: '<S44>/Logical Operator1'
   *  Logic: '<S44>/Logical Operator2'
   *  Logic: '<S44>/Logical Operator7'
   *  MATLAB Function: '<S8>/MATLAB Function'
   *  RelationalOperator: '<S44>/Equal'
   *  RelationalOperator: '<S44>/Relational Operator'
   *  RelationalOperator: '<S44>/Relational Operator1'
   *  Signum: '<S44>/Sign1'
   *  Signum: '<S44>/Sign2'
   */
  rtb_LogicalOperator_f = (((rtb_Sum2_e >= rtb_Switch7) || (rtb_Sum2_e <=
    rtb_Switch6)) && ((rtb_Sum2_e_0 == tmp_2) || (!bCtrl_enable)));

  /* BusCreator: '<S5>/Bus Creator1' incorporates:
   *  BusCreator: '<S8>/Bus Creator'
   *  MATLAB Function: '<S8>/MATLAB Function'
   */
  LX2_Y.tLX2_DBUG_j.Stm.rP_act_Norm_Filt = LX2_B.Filter1_i.Switch;
  LX2_Y.tLX2_DBUG_j.Stm.bBPOC_enable[0] = rtb_bBPOC_enable_a[0];
  LX2_Y.tLX2_DBUG_j.Stm.bBPOC_enable[1] = rtb_bBPOC_enable_a[1];
  LX2_Y.tLX2_DBUG_j.Stm.bBPOC_enable[2] = rtb_bBPOC_enable_a[2];
  LX2_Y.tLX2_DBUG_j.Stm.bBPOC_enable[3] = rtb_bBPOC_enable_a[3];
  LX2_Y.tLX2_DBUG_j.Stm.bBPOC_save_enable[0] = rtb_bSave_BPOC_enable[0];
  LX2_Y.tLX2_DBUG_j.Stm.bBPOC_save_enable[1] = rtb_bSave_BPOC_enable[1];
  LX2_Y.tLX2_DBUG_j.Stm.bBPOC_save_enable[2] = rtb_bSave_BPOC_enable[2];
  LX2_Y.tLX2_DBUG_j.Stm.bBPOC_save_enable[3] = rtb_bSave_BPOC_enable[3];
  LX2_Y.tLX2_DBUG_j.Stm.rSplitfactor_Gas[0] = rtb_splitfactor_Gas[0];
  LX2_Y.tLX2_DBUG_j.Stm.rSplitfactor_Gas[1] = rtb_splitfactor_Gas[1];
  LX2_Y.tLX2_DBUG_j.Stm.rSplitfactor_Gas[2] = rtb_splitfactor_Gas[2];
  LX2_Y.tLX2_DBUG_j.Stm.rSplitfactor_Gas[3] = rtb_splitfactor_Gas[3];
  LX2_Y.tLX2_DBUG_j.Stm.bCtrl_enable = bCtrl_enable;
  LX2_Y.tLX2_DBUG_j.Stm.bCtrl_freeze = bCtrl_freeze;
  LX2_Y.tLX2_DBUG_j.Stm.bEng_knock = b_bEng_knock;
  LX2_Y.tLX2_DBUG_j.Stm.bEng_misfire = bEng_misfire;
  LX2_Y.tLX2_DBUG_j.Stm.bBPOC_reset = rtb_LogicalOperator5_k;

  /* DataTypeConversion: '<S54>/Data Type Conversion1' */
  tmp_1 = (real32_T)fmod((real32_T)floor(LX2_B.TON_p.DiscreteTimeIntegrator),
    65536.0F);

  /* BusCreator: '<S5>/Bus Creator1' incorporates:
   *  BusCreator: '<S10>/Bus Creator1'
   *  BusCreator: '<S11>/Bus Creator1'
   *  BusCreator: '<S12>/Bus Creator1'
   *  BusCreator: '<S13>/Bus Creator1'
   *  BusCreator: '<S7>/Bus Creator1'
   *  BusCreator: '<S8>/Bus Creator'
   *  DataTypeConversion: '<S54>/Data Type Conversion1'
   *  Logic: '<S9>/Logical Operator'
   *  MATLAB Function: '<S7>/MATLAB Function'
   *  Product: '<S9>/Product'
   *  Product: '<S9>/Product1'
   *  Product: '<S9>/Product2'
   *  Product: '<S9>/Product3'
   *  Product: '<S9>/Product4'
   *  Product: '<S9>/Product5'
   *  Product: '<S9>/Product6'
   *  Product: '<S9>/Product7'
   *  Selector: '<S10>/Selector3'
   *  Selector: '<S11>/Selector3'
   *  Selector: '<S12>/Selector3'
   *  Selector: '<S13>/Selector3'
   *  Selector: '<S9>/Selector1'
   *  Selector: '<S9>/Selector16'
   *  Selector: '<S9>/Selector17'
   *  Selector: '<S9>/Selector18'
   *  Selector: '<S9>/Selector19'
   *  Selector: '<S9>/Selector2'
   *  Selector: '<S9>/Selector3'
   *  Selector: '<S9>/Selector4'
   *  Sum: '<S9>/Add'
   *  Sum: '<S9>/Sum of Elements'
   *  Sum: '<S9>/Sum of Elements1'
   *  Sum: '<S9>/Sum of Elements2'
   */
  LX2_Y.tLX2_DBUG_j.Stm.iTimer_save = (uint16_T)(tmp_1 < 0.0F ? (uint16_T)
    (int32_T)(int16_T)-(int16_T)(uint16_T)-tmp_1 : (uint16_T)tmp_1);
  LX2_Y.tLX2_DBUG_j.Stm.bLX2_SteadyState = rtb_LogicalOperator3_e;
  LX2_Y.tLX2_DBUG_j.Stm.bLX2_SteadyState_noDelay = rtb_LogicalOperator2;
  LX2_Y.tLX2_DBUG_j.Stm.bLX2_LeanoxDev_Steady = rtb_u;
  LX2_Y.tLX2_DBUG_j.Stm.bLX2_P_Set_Steady = rtb_u_b;
  LX2_Y.tLX2_DBUG_j.Ctr.rCtrlError = rtb_Switch2_l;
  LX2_Y.tLX2_DBUG_j.Ctr.rPr_offset_Ctrl = rtb_DiscreteTimeIntegrator;
  LX2_Y.tLX2_DBUG_j.Ctr.rPr_LX2_offset_preSat = rtb_Sum2_e;
  LX2_Y.tLX2_DBUG_j.Ctr.bLX2_inSaturation = rtb_LogicalOperator_f;
  LX2_Y.tLX2_DBUG_j.Ctr.rNOx_act_filt = rtb_splitfactor_VISU_idx;
  LX2_Y.tLX2_DBUG_j.Ctr.rPr_Ctrl_LowerLim_act = rtb_Switch6;
  LX2_Y.tLX2_DBUG_j.Ctr.rPr_Ctrl_UpperLim_act = rtb_Switch7;
  LX2_Y.tLX2_DBUG_j.Ctr.rPr_offset_BPOC_all = rtb_SumofElements;
  LX2_Y.tLX2_DBUG_j.Ctr.rPr_y0_Ctrl = b_y;
  LX2_Y.tLX2_DBUG_j.Ctr.rLX2_inLimit_Timer = LX2_B.TON_b.DiscreteTimeIntegrator;
  LX2_Y.tLX2_DBUG_j.Ctr.bLX2_inLimit_NoDelay = rtb_LogicalOperator4_g;
  LX2_Y.tLX2_DBUG_j.Gas1.bBPOC_enable = rtb_bBPOC_enable_a[0];
  LX2_Y.tLX2_DBUG_j.Gas1.bBPOC_save_enable = rtb_LogicalOperator7_m;
  for (i = 0; i < 11; i++) {
    LX2_Y.tLX2_DBUG_j.Gas1.bBPOC_measured_map_IN[i] = rtb_Delay1[i];
    LX2_Y.tLX2_DBUG_j.Gas1.rBPOC_offset_map_IN[i] = rtb_Delay2[i];
  }

  LX2_Y.tLX2_DBUG_j.Gas1.rPr_BPOC_offset_IN = rtb_Sum1;
  for (i = 0; i < 11; i++) {
    LX2_Y.tLX2_DBUG_j.Gas1.bBPOC_measured_map_OUT[i] =
      LX2_B.sf_BoostPressureOffsetCurve.OUT_measured[i];
    LX2_Y.tLX2_DBUG_j.Gas1.rBPOC_offset_map_OUT[i] = rtb_Switch2[i];
  }

  LX2_Y.tLX2_DBUG_j.Gas1.rPr_BPOC_offset_OUT = rtb_Switch3;
  LX2_Y.tLX2_DBUG_j.Gas1.rP_act_Norm_Filt = LX2_B.Filter1_i.Switch;
  LX2_Y.tLX2_DBUG_j.Gas1.rLX2_BPOC_Error = LX2_B.sf_BoostPressureOffsetCurve.e;
  LX2_Y.tLX2_DBUG_j.Gas1.rLX2_Lp[0] = rtb_Lp2Lp3Lp_c[0];
  LX2_Y.tLX2_DBUG_j.Gas1.rLX2_Lp[1] = rtb_Lp2Lp3Lp_c[1];
  LX2_Y.tLX2_DBUG_j.Gas1.rLX2_Lp[2] = rtb_Lp2Lp3Lp_c[2];
  LX2_Y.tLX2_DBUG_j.Gas1.rBPOC_DBUG_a[0] =
    LX2_B.sf_BoostPressureOffsetCurve.DBUG_a[0];
  LX2_Y.tLX2_DBUG_j.Gas1.rBPOC_DBUG_a[1] =
    LX2_B.sf_BoostPressureOffsetCurve.DBUG_a[1];
  LX2_Y.tLX2_DBUG_j.Gas1.rBPOC_DBUG_b[0] =
    LX2_B.sf_BoostPressureOffsetCurve.DBUG_b[0];
  LX2_Y.tLX2_DBUG_j.Gas1.rBPOC_DBUG_b[1] =
    LX2_B.sf_BoostPressureOffsetCurve.DBUG_b[1];
  LX2_Y.tLX2_DBUG_j.Gas1.rBPOC_DBUG_Lp[0] =
    LX2_B.sf_BoostPressureOffsetCurve.DBUG_Lp[0];
  LX2_Y.tLX2_DBUG_j.Gas1.rBPOC_DBUG_Lp[1] =
    LX2_B.sf_BoostPressureOffsetCurve.DBUG_Lp[1];
  LX2_Y.tLX2_DBUG_j.Gas1.rBPOC_DBUG_Lp[2] =
    LX2_B.sf_BoostPressureOffsetCurve.DBUG_Lp[2];
  LX2_Y.tLX2_DBUG_j.Gas1.rBPOC_DBUG_Lp[3] =
    LX2_B.sf_BoostPressureOffsetCurve.DBUG_Lp[3];
  LX2_Y.tLX2_DBUG_j.Gas1.rBPOC_DBUG_s[0] =
    LX2_B.sf_BoostPressureOffsetCurve.DBUG_s[0];
  LX2_Y.tLX2_DBUG_j.Gas1.rBPOC_DBUG_s[1] =
    LX2_B.sf_BoostPressureOffsetCurve.DBUG_s[1];
  LX2_Y.tLX2_DBUG_j.Gas1.rBPOC_DBUG_s[2] =
    LX2_B.sf_BoostPressureOffsetCurve.DBUG_s[2];
  LX2_Y.tLX2_DBUG_j.Gas2.bBPOC_enable = rtb_bBPOC_enable_a[1];
  LX2_Y.tLX2_DBUG_j.Gas2.bBPOC_save_enable = rtb_LogicalOperator7_e;
  for (i = 0; i < 11; i++) {
    LX2_Y.tLX2_DBUG_j.Gas2.bBPOC_measured_map_IN[i] = rtb_Delay1_g[i];
    LX2_Y.tLX2_DBUG_j.Gas2.rBPOC_offset_map_IN[i] = rtb_Delay2_e[i];
  }

  LX2_Y.tLX2_DBUG_j.Gas2.rPr_BPOC_offset_IN = rtb_Sum1_e;
  for (i = 0; i < 11; i++) {
    LX2_Y.tLX2_DBUG_j.Gas2.bBPOC_measured_map_OUT[i] =
      LX2_B.sf_BoostPressureOffsetCurve_f.OUT_measured[i];
    LX2_Y.tLX2_DBUG_j.Gas2.rBPOC_offset_map_OUT[i] = rtb_Switch2_j[i];
  }

  LX2_Y.tLX2_DBUG_j.Gas2.rPr_BPOC_offset_OUT = rtb_SumofElements2;
  LX2_Y.tLX2_DBUG_j.Gas2.rP_act_Norm_Filt = LX2_B.Filter1_i.Switch;
  LX2_Y.tLX2_DBUG_j.Gas2.rLX2_BPOC_Error = LX2_B.sf_BoostPressureOffsetCurve_f.e;
  LX2_Y.tLX2_DBUG_j.Gas2.rLX2_Lp[0] = rtb_Lp2Lp3Lp_c_n[0];
  LX2_Y.tLX2_DBUG_j.Gas2.rLX2_Lp[1] = rtb_Lp2Lp3Lp_c_n[1];
  LX2_Y.tLX2_DBUG_j.Gas2.rLX2_Lp[2] = rtb_Lp2Lp3Lp_c_n[2];
  LX2_Y.tLX2_DBUG_j.Gas2.rBPOC_DBUG_a[0] =
    LX2_B.sf_BoostPressureOffsetCurve_f.DBUG_a[0];
  LX2_Y.tLX2_DBUG_j.Gas2.rBPOC_DBUG_a[1] =
    LX2_B.sf_BoostPressureOffsetCurve_f.DBUG_a[1];
  LX2_Y.tLX2_DBUG_j.Gas2.rBPOC_DBUG_b[0] =
    LX2_B.sf_BoostPressureOffsetCurve_f.DBUG_b[0];
  LX2_Y.tLX2_DBUG_j.Gas2.rBPOC_DBUG_b[1] =
    LX2_B.sf_BoostPressureOffsetCurve_f.DBUG_b[1];
  LX2_Y.tLX2_DBUG_j.Gas2.rBPOC_DBUG_Lp[0] =
    LX2_B.sf_BoostPressureOffsetCurve_f.DBUG_Lp[0];
  LX2_Y.tLX2_DBUG_j.Gas2.rBPOC_DBUG_Lp[1] =
    LX2_B.sf_BoostPressureOffsetCurve_f.DBUG_Lp[1];
  LX2_Y.tLX2_DBUG_j.Gas2.rBPOC_DBUG_Lp[2] =
    LX2_B.sf_BoostPressureOffsetCurve_f.DBUG_Lp[2];
  LX2_Y.tLX2_DBUG_j.Gas2.rBPOC_DBUG_Lp[3] =
    LX2_B.sf_BoostPressureOffsetCurve_f.DBUG_Lp[3];
  LX2_Y.tLX2_DBUG_j.Gas2.rBPOC_DBUG_s[0] =
    LX2_B.sf_BoostPressureOffsetCurve_f.DBUG_s[0];
  LX2_Y.tLX2_DBUG_j.Gas2.rBPOC_DBUG_s[1] =
    LX2_B.sf_BoostPressureOffsetCurve_f.DBUG_s[1];
  LX2_Y.tLX2_DBUG_j.Gas2.rBPOC_DBUG_s[2] =
    LX2_B.sf_BoostPressureOffsetCurve_f.DBUG_s[2];
  LX2_Y.tLX2_DBUG_j.Gas3.bBPOC_enable = rtb_bBPOC_enable_a[2];
  LX2_Y.tLX2_DBUG_j.Gas3.bBPOC_save_enable = rtb_LogicalOperator7_l;
  for (i = 0; i < 11; i++) {
    LX2_Y.tLX2_DBUG_j.Gas3.bBPOC_measured_map_IN[i] = rtb_Delay1_l[i];
    LX2_Y.tLX2_DBUG_j.Gas3.rBPOC_offset_map_IN[i] = rtb_Delay2_o[i];
  }

  LX2_Y.tLX2_DBUG_j.Gas3.rPr_BPOC_offset_IN = rtb_Sum1_b;
  for (i = 0; i < 11; i++) {
    LX2_Y.tLX2_DBUG_j.Gas3.bBPOC_measured_map_OUT[i] =
      LX2_B.sf_BoostPressureOffsetCurve_d.OUT_measured[i];
    LX2_Y.tLX2_DBUG_j.Gas3.rBPOC_offset_map_OUT[i] = rtb_Switch2_k[i];
  }

  LX2_Y.tLX2_DBUG_j.Gas3.rPr_BPOC_offset_OUT = rtb_SumofElements1;
  LX2_Y.tLX2_DBUG_j.Gas3.rP_act_Norm_Filt = LX2_B.Filter1_i.Switch;
  LX2_Y.tLX2_DBUG_j.Gas3.rLX2_BPOC_Error = LX2_B.sf_BoostPressureOffsetCurve_d.e;
  LX2_Y.tLX2_DBUG_j.Gas3.rLX2_Lp[0] = rtb_Lp2Lp3Lp_c_l[0];
  LX2_Y.tLX2_DBUG_j.Gas3.rLX2_Lp[1] = rtb_Lp2Lp3Lp_c_l[1];
  LX2_Y.tLX2_DBUG_j.Gas3.rLX2_Lp[2] = rtb_Lp2Lp3Lp_c_l[2];
  LX2_Y.tLX2_DBUG_j.Gas3.rBPOC_DBUG_a[0] =
    LX2_B.sf_BoostPressureOffsetCurve_d.DBUG_a[0];
  LX2_Y.tLX2_DBUG_j.Gas3.rBPOC_DBUG_a[1] =
    LX2_B.sf_BoostPressureOffsetCurve_d.DBUG_a[1];
  LX2_Y.tLX2_DBUG_j.Gas3.rBPOC_DBUG_b[0] =
    LX2_B.sf_BoostPressureOffsetCurve_d.DBUG_b[0];
  LX2_Y.tLX2_DBUG_j.Gas3.rBPOC_DBUG_b[1] =
    LX2_B.sf_BoostPressureOffsetCurve_d.DBUG_b[1];
  LX2_Y.tLX2_DBUG_j.Gas3.rBPOC_DBUG_Lp[0] =
    LX2_B.sf_BoostPressureOffsetCurve_d.DBUG_Lp[0];
  LX2_Y.tLX2_DBUG_j.Gas3.rBPOC_DBUG_Lp[1] =
    LX2_B.sf_BoostPressureOffsetCurve_d.DBUG_Lp[1];
  LX2_Y.tLX2_DBUG_j.Gas3.rBPOC_DBUG_Lp[2] =
    LX2_B.sf_BoostPressureOffsetCurve_d.DBUG_Lp[2];
  LX2_Y.tLX2_DBUG_j.Gas3.rBPOC_DBUG_Lp[3] =
    LX2_B.sf_BoostPressureOffsetCurve_d.DBUG_Lp[3];
  LX2_Y.tLX2_DBUG_j.Gas3.rBPOC_DBUG_s[0] =
    LX2_B.sf_BoostPressureOffsetCurve_d.DBUG_s[0];
  LX2_Y.tLX2_DBUG_j.Gas3.rBPOC_DBUG_s[1] =
    LX2_B.sf_BoostPressureOffsetCurve_d.DBUG_s[1];
  LX2_Y.tLX2_DBUG_j.Gas3.rBPOC_DBUG_s[2] =
    LX2_B.sf_BoostPressureOffsetCurve_d.DBUG_s[2];
  LX2_Y.tLX2_DBUG_j.Gas4.bBPOC_enable = rtb_bBPOC_enable_a[3];
  LX2_Y.tLX2_DBUG_j.Gas4.bBPOC_save_enable = rtb_LogicalOperator7_i;
  for (i = 0; i < 11; i++) {
    LX2_Y.tLX2_DBUG_j.Gas4.bBPOC_measured_map_IN[i] = rtb_Delay1_c[i];
    LX2_Y.tLX2_DBUG_j.Gas4.rBPOC_offset_map_IN[i] = rtb_Delay2_o1[i];
  }

  LX2_Y.tLX2_DBUG_j.Gas4.rPr_BPOC_offset_IN = rtb_Sum1_h;
  for (i = 0; i < 11; i++) {
    LX2_Y.tLX2_DBUG_j.Gas4.bBPOC_measured_map_OUT[i] =
      LX2_B.sf_BoostPressureOffsetCurve_a.OUT_measured[i];
    LX2_Y.tLX2_DBUG_j.Gas4.rBPOC_offset_map_OUT[i] = rtb_Switch2_kq[i];
  }

  LX2_Y.tLX2_DBUG_j.Gas4.rPr_BPOC_offset_OUT = rtb_SumofElements_o;
  LX2_Y.tLX2_DBUG_j.Gas4.rP_act_Norm_Filt = LX2_B.Filter1_i.Switch;
  LX2_Y.tLX2_DBUG_j.Gas4.rLX2_BPOC_Error = LX2_B.sf_BoostPressureOffsetCurve_a.e;
  LX2_Y.tLX2_DBUG_j.Gas4.rLX2_Lp[0] = rtb_Lp2Lp3Lp_c_e[0];
  LX2_Y.tLX2_DBUG_j.Gas4.rLX2_Lp[1] = rtb_Lp2Lp3Lp_c_e[1];
  LX2_Y.tLX2_DBUG_j.Gas4.rLX2_Lp[2] = rtb_Lp2Lp3Lp_c_e[2];
  LX2_Y.tLX2_DBUG_j.Gas4.rBPOC_DBUG_a[0] =
    LX2_B.sf_BoostPressureOffsetCurve_a.DBUG_a[0];
  LX2_Y.tLX2_DBUG_j.Gas4.rBPOC_DBUG_a[1] =
    LX2_B.sf_BoostPressureOffsetCurve_a.DBUG_a[1];
  LX2_Y.tLX2_DBUG_j.Gas4.rBPOC_DBUG_b[0] =
    LX2_B.sf_BoostPressureOffsetCurve_a.DBUG_b[0];
  LX2_Y.tLX2_DBUG_j.Gas4.rBPOC_DBUG_b[1] =
    LX2_B.sf_BoostPressureOffsetCurve_a.DBUG_b[1];
  LX2_Y.tLX2_DBUG_j.Gas4.rBPOC_DBUG_Lp[0] =
    LX2_B.sf_BoostPressureOffsetCurve_a.DBUG_Lp[0];
  LX2_Y.tLX2_DBUG_j.Gas4.rBPOC_DBUG_Lp[1] =
    LX2_B.sf_BoostPressureOffsetCurve_a.DBUG_Lp[1];
  LX2_Y.tLX2_DBUG_j.Gas4.rBPOC_DBUG_Lp[2] =
    LX2_B.sf_BoostPressureOffsetCurve_a.DBUG_Lp[2];
  LX2_Y.tLX2_DBUG_j.Gas4.rBPOC_DBUG_Lp[3] =
    LX2_B.sf_BoostPressureOffsetCurve_a.DBUG_Lp[3];
  LX2_Y.tLX2_DBUG_j.Gas4.rBPOC_DBUG_s[0] =
    LX2_B.sf_BoostPressureOffsetCurve_a.DBUG_s[0];
  LX2_Y.tLX2_DBUG_j.Gas4.rBPOC_DBUG_s[1] =
    LX2_B.sf_BoostPressureOffsetCurve_a.DBUG_s[1];
  LX2_Y.tLX2_DBUG_j.Gas4.rBPOC_DBUG_s[2] =
    LX2_B.sf_BoostPressureOffsetCurve_a.DBUG_s[2];
  for (i = 0; i < 11; i++) {
    /* Switch: '<S9>/Switch21' incorporates:
     *  Constant: '<S9>/Constant17'
     *  Selector: '<S9>/Selector1'
     */
    if (rtb_splitfactor_Gas[0] != 0.0F) {
      rtb_splitfactor_VISU_idx = rtb_Switch2[i];
    } else {
      rtb_splitfactor_VISU_idx = 0.0F;
    }

    /* End of Switch: '<S9>/Switch21' */

    /* Switch: '<S9>/Switch1' incorporates:
     *  Constant: '<S9>/Constant2'
     *  Selector: '<S9>/Selector2'
     */
    if (rtb_splitfactor_Gas[1] != 0.0F) {
      rtb_UnitDelay3 = rtb_Switch2_j[i];
    } else {
      rtb_UnitDelay3 = 0.0F;
    }

    /* End of Switch: '<S9>/Switch1' */

    /* Switch: '<S9>/Switch2' incorporates:
     *  Constant: '<S9>/Constant4'
     *  Selector: '<S9>/Selector3'
     */
    if (rtb_splitfactor_Gas[2] != 0.0F) {
      rtb_UnitDelay2 = rtb_Switch2_k[i];
    } else {
      rtb_UnitDelay2 = 0.0F;
    }

    /* End of Switch: '<S9>/Switch2' */

    /* Switch: '<S9>/Switch3' incorporates:
     *  Constant: '<S9>/Constant6'
     *  Selector: '<S9>/Selector4'
     */
    if (rtb_splitfactor_Gas[3] != 0.0F) {
      rtb_Gain3 = rtb_Switch2_kq[i];
    } else {
      rtb_Gain3 = 0.0F;
    }

    /* End of Switch: '<S9>/Switch3' */
    LX2_Y.tLX2_DBUG_j.rLX2_BPOC_internal[i] = ((rtb_splitfactor_Gas[0] *
      rtb_splitfactor_VISU_idx + rtb_splitfactor_Gas[1] * rtb_UnitDelay3) +
      rtb_splitfactor_Gas[2] * rtb_UnitDelay2) + rtb_splitfactor_Gas[3] *
      rtb_Gain3;

    /* Switch: '<S9>/Switch6' incorporates:
     *  Constant: '<S9>/Constant7'
     *  Product: '<S9>/Product4'
     *  Product: '<S9>/Product5'
     *  Product: '<S9>/Product6'
     *  Product: '<S9>/Product7'
     *  Selector: '<S9>/Selector1'
     *  Selector: '<S9>/Selector2'
     *  Selector: '<S9>/Selector3'
     *  Selector: '<S9>/Selector4'
     *  Selector: '<S9>/Selector5'
     *  Sum: '<S9>/Add'
     */
    if (rtb_splitfactor_Gas[0] != 0.0F) {
      rtb_splitfactor_Gas_0 = (int32_T)
        LX2_B.sf_BoostPressureOffsetCurve.OUT_measured[i];
    } else {
      rtb_splitfactor_Gas_0 = 0;
    }

    /* End of Switch: '<S9>/Switch6' */

    /* Switch: '<S9>/Switch4' incorporates:
     *  Constant: '<S9>/Constant10'
     *  Selector: '<S9>/Selector6'
     */
    if (rtb_splitfactor_Gas[1] != 0.0F) {
      rtb_splitfactor_Gas_1 = (int32_T)
        LX2_B.sf_BoostPressureOffsetCurve_f.OUT_measured[i];
    } else {
      rtb_splitfactor_Gas_1 = 0;
    }

    /* End of Switch: '<S9>/Switch4' */

    /* Switch: '<S9>/Switch5' incorporates:
     *  Constant: '<S9>/Constant11'
     *  Selector: '<S9>/Selector7'
     */
    if (rtb_splitfactor_Gas[2] != 0.0F) {
      rtb_splitfactor_Gas_2 = (int32_T)
        LX2_B.sf_BoostPressureOffsetCurve_d.OUT_measured[i];
    } else {
      rtb_splitfactor_Gas_2 = 0;
    }

    /* End of Switch: '<S9>/Switch5' */

    /* Switch: '<S9>/Switch7' incorporates:
     *  Constant: '<S9>/Constant13'
     *  Selector: '<S9>/Selector8'
     */
    if (rtb_splitfactor_Gas[3] != 0.0F) {
      rtb_splitfactor_Gas_3 = (int32_T)
        LX2_B.sf_BoostPressureOffsetCurve_a.OUT_measured[i];
    } else {
      rtb_splitfactor_Gas_3 = 0;
    }

    /* End of Switch: '<S9>/Switch7' */
    LX2_Y.tLX2_DBUG_j.bLX2_BPOC_measured_internal[i] = ((rtb_splitfactor_Gas_0
      != 0) || (rtb_splitfactor_Gas_1 != 0) || (rtb_splitfactor_Gas_2 != 0) ||
      (rtb_splitfactor_Gas_3 != 0));
  }

  LX2_Y.tLX2_DBUG_j.rBPOC_Lp_all[0] = ((rtb_splitfactor_Gas[0] *
    LX2_B.sf_BoostPressureOffsetCurve.DBUG_Lp[1] + rtb_splitfactor_Gas[1] *
    LX2_B.sf_BoostPressureOffsetCurve_f.DBUG_Lp[1]) + rtb_splitfactor_Gas[2] *
    LX2_B.sf_BoostPressureOffsetCurve_d.DBUG_Lp[1]) + rtb_splitfactor_Gas[3] *
    LX2_B.sf_BoostPressureOffsetCurve_a.DBUG_Lp[1];
  LX2_Y.tLX2_DBUG_j.rBPOC_Lp_all[1] = ((rtb_splitfactor_Gas[0] *
    LX2_B.sf_BoostPressureOffsetCurve.DBUG_Lp[2] + rtb_splitfactor_Gas[1] *
    LX2_B.sf_BoostPressureOffsetCurve_f.DBUG_Lp[2]) + rtb_splitfactor_Gas[2] *
    LX2_B.sf_BoostPressureOffsetCurve_d.DBUG_Lp[2]) + rtb_splitfactor_Gas[3] *
    LX2_B.sf_BoostPressureOffsetCurve_a.DBUG_Lp[2];
  LX2_Y.tLX2_DBUG_j.rBPOC_Lp_all[2] = ((rtb_splitfactor_Gas[0] *
    LX2_B.sf_BoostPressureOffsetCurve.DBUG_Lp[3] + rtb_splitfactor_Gas[1] *
    LX2_B.sf_BoostPressureOffsetCurve_f.DBUG_Lp[3]) + rtb_splitfactor_Gas[2] *
    LX2_B.sf_BoostPressureOffsetCurve_d.DBUG_Lp[3]) + rtb_splitfactor_Gas[3] *
    LX2_B.sf_BoostPressureOffsetCurve_a.DBUG_Lp[3];

  /* S-Function (bur_bus_out): '<Root>/Bus Output' */
  inst->Output = LX2_Y.tLX2_OUT_c;

  /* S-Function (bur_bus_out): '<Root>/Bus Output1' */
  inst->DBUG = LX2_Y.tLX2_DBUG_j;

  /* Switch: '<S36>/Switch' incorporates:
   *  Constant: '<S36>/Constant'
   */
  if (rtb_LogicalOperator_f) {
    rtb_UnitDelay3 = 0.0F;
  } else {
    rtb_UnitDelay3 = rtb_Divide;
  }

  /* End of Switch: '<S36>/Switch' */

  /* UnitDelay: '<S4>/Unit Delay' */
  LX2_B.UnitDelay = LX2_DWork.UnitDelay_DSTATE;

  /* S-Function (bur_out): '<Root>/Output' */
  inst->Version = LX2_B.UnitDelay;

  /* Update for UnitDelay: '<S7>/Unit Delay3' */
  LX2_DWork.UnitDelay3_DSTATE = rtb_Switch2_kt;

  /* Update for UnitDelay: '<S7>/Unit Delay1' */
  LX2_DWork.UnitDelay1_DSTATE = rtb_Compare_n;

  /* Update for UnitDelay: '<S52>/Unit Delay1' */
  LX2_DWork.UnitDelay1_DSTATE_l = rtb_Compare_n;

  /* Update for UnitDelay: '<S54>/Unit Delay' */
  LX2_DWork.UnitDelay_DSTATE_l = LX2_B.TON_p.LogicalOperator3;

  /* Update for Delay: '<S10>/Delay2' */
  LX2_DWork.icLoad = 0U;

  /* Update for UnitDelay: '<S6>/Unit Delay2' */
  LX2_DWork.UnitDelay2_DSTATE = rtb_Switch2_kt;

  /* Update for Delay: '<S10>/Delay1' */
  LX2_DWork.icLoad_o = 0U;

  /* Update for Delay: '<S11>/Delay2' */
  LX2_DWork.icLoad_or = 0U;

  /* Update for Delay: '<S11>/Delay1' */
  LX2_DWork.icLoad_oj = 0U;

  /* Update for Delay: '<S12>/Delay2' */
  LX2_DWork.icLoad_p = 0U;

  /* Update for Delay: '<S12>/Delay1' */
  LX2_DWork.icLoad_d = 0U;

  /* Update for Delay: '<S13>/Delay2' */
  LX2_DWork.icLoad_f = 0U;

  /* Update for Delay: '<S13>/Delay1' */
  LX2_DWork.icLoad_c = 0U;
  for (i = 0; i < 11; i++) {
    /* Update for Delay: '<S10>/Delay2' */
    LX2_DWork.Delay2_DSTATE[i] = rtb_Switch2[i];

    /* Update for Delay: '<S10>/Delay1' */
    LX2_DWork.Delay1_DSTATE[i] =
      LX2_B.sf_BoostPressureOffsetCurve.OUT_measured[i];

    /* Update for Delay: '<S11>/Delay2' */
    LX2_DWork.Delay2_DSTATE_j[i] = rtb_Switch2_j[i];

    /* Update for Delay: '<S11>/Delay1' */
    LX2_DWork.Delay1_DSTATE_l[i] =
      LX2_B.sf_BoostPressureOffsetCurve_f.OUT_measured[i];

    /* Update for Delay: '<S12>/Delay2' */
    LX2_DWork.Delay2_DSTATE_b[i] = rtb_Switch2_k[i];

    /* Update for Delay: '<S12>/Delay1' */
    LX2_DWork.Delay1_DSTATE_o[i] =
      LX2_B.sf_BoostPressureOffsetCurve_d.OUT_measured[i];

    /* Update for Delay: '<S13>/Delay2' */
    LX2_DWork.Delay2_DSTATE_d[i] = rtb_Switch2_kq[i];
    LX2_DWork.Delay1_DSTATE_g[i] =
      LX2_B.sf_BoostPressureOffsetCurve_a.OUT_measured[i];
  }

  /* End of Update for Delay: '<S13>/Delay1' */

  /* Update for UnitDelay: '<S7>/Unit Delay5' */
  LX2_DWork.UnitDelay5_DSTATE = rtb_SumofElements;

  /* Update for UnitDelay: '<S7>/Unit Delay6' */
  LX2_DWork.UnitDelay6_DSTATE = rtb_DiscreteTimeIntegrator;

  /* Update for DiscreteIntegrator: '<S36>/Discrete-Time Integrator' */
  LX2_DWork.DiscreteTimeIntegrator_IC_LOADI = 0U;
  LX2_DWork.DiscreteTimeIntegrator_DSTATE += 0.000100000005F * rtb_UnitDelay3;
  if (rtb_Reset) {
    LX2_DWork.DiscreteTimeIntegrator_PrevRese = 1;
  } else {
    LX2_DWork.DiscreteTimeIntegrator_PrevRese = 0;
  }

  /* End of Update for DiscreteIntegrator: '<S36>/Discrete-Time Integrator' */

  /* Update for UnitDelay: '<S7>/Unit Delay4' */
  LX2_DWork.UnitDelay4_DSTATE = rtb_Switch2_kt;

  /* Update for Delay: '<S41>/Delay' */
  LX2_DWork.icLoad_i = 0U;
  LX2_DWork.Delay_DSTATE = rtb_Switch2_kt;

  /* Update for UnitDelay: '<S34>/Delay Input1' */
  LX2_DWork.DelayInput1_DSTATE = LX2_B.BusInput.bNOx_valid;

  /* Update for UnitDelay: '<S4>/Unit Delay' */
  LX2_DWork.UnitDelay_DSTATE = 130U;
}

/* Model initialize function */
void LX2_initialize(struct fLX2* inst)
{
  LX2_PrevZCSigState.Delay2_Reset_ZCE = UNINITIALIZED_ZCSIG;
  LX2_PrevZCSigState.Delay1_Reset_ZCE = UNINITIALIZED_ZCSIG;
  LX2_PrevZCSigState.Delay2_Reset_ZCE_o = UNINITIALIZED_ZCSIG;
  LX2_PrevZCSigState.Delay1_Reset_ZCE_n = UNINITIALIZED_ZCSIG;
  LX2_PrevZCSigState.Delay2_Reset_ZCE_or = UNINITIALIZED_ZCSIG;
  LX2_PrevZCSigState.Delay1_Reset_ZCE_e = UNINITIALIZED_ZCSIG;
  LX2_PrevZCSigState.Delay2_Reset_ZCE_k = UNINITIALIZED_ZCSIG;
  LX2_PrevZCSigState.Delay1_Reset_ZCE_k = UNINITIALIZED_ZCSIG;
  LX2_PrevZCSigState.Delay_Reset_ZCE = UNINITIALIZED_ZCSIG;

  /* InitializeConditions for Atomic SubSystem: '<S51>/Filter' */
  LX2_Filter1_Init(&LX2_DWork.Filter, inst);

  /* End of InitializeConditions for SubSystem: '<S51>/Filter' */

  /* InitializeConditions for Atomic SubSystem: '<S51>/Filter1' */
  LX2_Filter1_Init(&LX2_DWork.Filter1, inst);

  /* End of InitializeConditions for SubSystem: '<S51>/Filter1' */

  /* InitializeConditions for Atomic SubSystem: '<S8>/Filter1' */
  LX2_Filter1_Init(&LX2_DWork.Filter1_i, inst);

  /* End of InitializeConditions for SubSystem: '<S8>/Filter1' */

  /* InitializeConditions for Delay: '<S10>/Delay2' */
  LX2_DWork.icLoad = 1U;

  /* InitializeConditions for Delay: '<S10>/Delay1' */
  LX2_DWork.icLoad_o = 1U;

  /* InitializeConditions for Delay: '<S11>/Delay2' */
  LX2_DWork.icLoad_or = 1U;

  /* InitializeConditions for Delay: '<S11>/Delay1' */
  LX2_DWork.icLoad_oj = 1U;

  /* InitializeConditions for Delay: '<S12>/Delay2' */
  LX2_DWork.icLoad_p = 1U;

  /* InitializeConditions for Delay: '<S12>/Delay1' */
  LX2_DWork.icLoad_d = 1U;

  /* InitializeConditions for Delay: '<S13>/Delay2' */
  LX2_DWork.icLoad_f = 1U;

  /* InitializeConditions for Delay: '<S13>/Delay1' */
  LX2_DWork.icLoad_c = 1U;

  /* InitializeConditions for DiscreteIntegrator: '<S36>/Discrete-Time Integrator' */
  LX2_DWork.DiscreteTimeIntegrator_IC_LOADI = 1U;

  /* InitializeConditions for Delay: '<S41>/Delay' */
  LX2_DWork.icLoad_i = 1U;

  /* InitializeConditions for Atomic SubSystem: '<S7>/Filter' */
  /* InitializeConditions for DiscreteIntegrator: '<S35>/Discrete-Time Integrator' */
  LX2_DWork.DiscreteTimeIntegrator_IC_LOA_l = 1U;

  /* End of InitializeConditions for SubSystem: '<S7>/Filter' */
}

/* Model terminate function */
void LX2_terminate(struct fLX2* inst)
{
  /* (no terminate code required) */
}

/*======================== TOOL VERSION INFORMATION ==========================*
 * MATLAB 8.0 (R2012b)20-Jul-2012                                             *
 * Simulink 8.0 (R2012b)20-Jul-2012                                           *
 * Simulink Coder 8.3 (R2012b)20-Jul-2012                                     *
 * Embedded Coder 6.3 (R2012b)20-Jul-2012                                     *
 * Stateflow 8.0 (R2012b)20-Jul-2012                                          *
 *============================================================================*/

/*======================= LICENSE IN USE INFORMATION =========================*
 * matlab                                                                     *
 * matlab_coder                                                               *
 * real-time_workshop                                                         *
 * rtw_embedded_coder                                                         *
 * simulink                                                                   *
 *============================================================================*/
```

#### LX2_data.c
```c
/********************************************************************
 * COPYRIGHT -- Bernecker + Rainer Industrie-Elektronik Ges.m.b.H.
 ********************************************************************
 * Program: LX2
 * File: LX2_data.c
 * Author: 212566120
 * Created: Wed Apr 11 13:34:17 2018
 ********************************************************************
 * Data for program LX2
 ********************************************************************
 * Generated with B&R Automation Studio Target for Simulink V4.2
 * (ERT based)
 ********************************************************************/
#include "LX2.h"
#include "LX2_private.h"

/*  GLOBAL DATA DEFINITIONS */

/* Constant parameters (auto storage) */
const ConstParam_LX2 LX2_ConstP = {
  /* Pooled Parameter (Expression: single(0:10:100))
   * Referenced by:
   *   '<S10>/Constant2'
   *   '<S11>/Constant2'
   *   '<S12>/Constant2'
   *   '<S13>/Constant2'
   */
  { 0.0F, 10.0F, 20.0F, 30.0F, 40.0F, 50.0F, 60.0F, 70.0F, 80.0F, 90.0F, 100.0F
  }
};
```

#### fLX2.c
```c
/********************************************************************
 * COPYRIGHT -- Bernecker + Rainer Industrie-Elektronik Ges.m.b.H.
 ********************************************************************
 * Program: LX2
 * File: fLX2.c
 * Author: 212566120
 * Created: Wed Apr 11 13:34:17 2018
 ********************************************************************
 * Implementation of program LX2
 ********************************************************************
 * Generated with B&R Automation Studio Target for Simulink V4.2
 * (ERT based)
 ********************************************************************/
#include <bur/plctypes.h>
#include "LX2.h"
#include "rtwtypes.h"

/* Defines */
#define SS_TERMINATE 4
#define SS_OUTPUT 3
#define SS_INITIALIZE 2

/*  Data Types */

/**************************** GLOBAL DATA *************************************/
/*  Definitions */

/*  Declarations  */

/***************************** FILE SCOPE DATA ********************************/

/*************************** FUNCTIONS ****************************************/
#ifdef __cplusplus

unsigned long bur_heap_size = 6553500;

#endif

void fLX2(struct fLX2* inst)
{

  switch (inst->ssMethodType)
  {
   case SS_INITIALIZE:
    /* call model initialize function */
    LX2_initialize(inst);
    break;

   case SS_OUTPUT:
    /* call model step function */
    LX2_step(inst);

    break;

   case SS_TERMINATE:
    /* call model terminate function */
    LX2_terminate(inst);
    break;
  }
}

/*****************************************************************************
   Function block sample time: 0.099999999999999992s
 *****************************************************************************/

/*****************************************************************************
   B&R Automation Studio Target for Simulink Version: A4.5.1 (27-Jul-2015)
 *****************************************************************************/

/*======================== TOOL VERSION INFORMATION ==========================*
 * MATLAB 8.0 (R2012b)20-Jul-2012                                             *
 * Simulink 8.0 (R2012b)20-Jul-2012                                           *
 * Simulink Coder 8.3 (R2012b)20-Jul-2012                                     *
 * Embedded Coder 6.3 (R2012b)20-Jul-2012                                     *
 * Stateflow 8.0 (R2012b)20-Jul-2012                                          *
 *============================================================================*/

/*======================= LICENSE IN USE INFORMATION =========================*
 * matlab                                                                     *
 * matlab_coder                                                               *
 * real-time_workshop                                                         *
 * rtw_embedded_coder                                                         *
 * simulink                                                                   *
 *============================================================================*/
```
